LIN {X 0,Y 218.653,Z 421.951,A -85,B 0,C 180,E1 -22546.919,E2 -22546.919} C_VEL
LIN {X 0,Y 215.686,Z 434.453,A -85,B 0,C 180,E1 -22548.088,E2 -22548.088} C_VEL
LIN {X 0,Y 212.005,Z 447.131,A -85,B 0,C 180,E1 -22549.628,E2 -22549.628} C_VEL
LIN {X 0,Y 207.893,Z 459.523,A -85,B 0,C 180,E1 -22551.597,E2 -22551.597} C_VEL
LIN {X 0,Y 203.913,Z 469.49,A -85,B 0,C 180,E1 -22553.52,E2 -22553.52} C_VEL
LIN {X 0,Y 199.074,Z 480.574,A -85,B 0,C 180,E1 -22556.218,E2 -22556.218} C_VEL
LIN {X 0,Y 194.639,Z 489.759,A -85,B 0,C 180,E1 -22559.033,E2 -22559.033} C_VEL
LIN {X 0,Y 190.05,Z 498.52,A -85,B 0,C 180,E1 -22562.422,E2 -22562.422} C_VEL
LIN {X 0,Y 186.885,Z 504.847,A -85,B 0,C 180,E1 -22565.564,E2 -22565.564} C_VEL
LIN {X 0,Y 182.861,Z 511.661,A -85,B 0,C 180,E1 -22569.763,E2 -22569.763} C_VEL
LIN {X 0,Y 180.074,Z 516.84,A -85,B 0,C 180,E1 -22574.145,E2 -22574.145} C_VEL
LIN {X 0,Y 178.099,Z 520.594,A -85,B 0,C 180,E1 -22578.62,E2 -22578.62} C_VEL
LIN {X 0,Y 176.962,Z 523.045,A -85,B 0,C 180,E1 -22583.157,E2 -22583.157} C_VEL
LIN {X 0,Y 176.433,Z 524.266,A -85,B 0,C 180,E1 -22587.716,E2 -22587.716} C_VEL
LIN {X 0,Y 176.423,Z 524.285,A -85,B 0,C 180,E1 -22592.282,E2 -22592.282} C_VEL
LIN {X 0,Y 176.901,Z 523.107,A -85,B 0,C 180,E1 -22596.844,E2 -22596.844} C_VEL
LIN {X 0,Y 178.034,Z 520.699,A -85,B 0,C 180,E1 -22601.383,E2 -22601.383} C_VEL
LIN {X 0,Y 180.021,Z 516.984,A -85,B 0,C 180,E1 -22605.858,E2 -22605.858} C_VEL
LIN {X 0,Y 182.79,Z 511.867,A -85,B 0,C 180,E1 -22610.244,E2 -22610.244} C_VEL
LIN {X 0,Y 185.684,Z 506.949,A -85,B 0,C 180,E1 -22613.416,E2 -22613.416} C_VEL
LIN {X 0,Y 189.292,Z 500.114,A -85,B 0,C 180,E1 -22616.992,E2 -22616.992} C_VEL
LIN {X 0,Y 193.801,Z 491.473,A -85,B 0,C 180,E1 -22620.509,E2 -22620.509} C_VEL
LIN {X 0,Y 198.243,Z 482.622,A -85,B 0,C 180,E1 -22623.331,E2 -22623.331} C_VEL
LIN {X 0,Y 202.955,Z 471.992,A -85,B 0,C 180,E1 -22626.062,E2 -22626.062} C_VEL
LIN {X 0,Y 207.337,Z 461.314,A -85,B 0,C 180,E1 -22628.213,E2 -22628.213} C_VEL
LIN {X 0,Y 211.244,Z 450.035,A -85,B 0,C 180,E1 -22630.075,E2 -22630.075} C_VEL
LIN {X 0,Y 215.079,Z 437.178,A -85,B 0,C 180,E1 -22631.741,E2 -22631.741} C_VEL
LIN {X 0,Y 218.486,Z 423.175,A -85,B 0,C 180,E1 -22633.12,E2 -22633.12} C_VEL
LIN {X 0,Y 221.137,Z 409.142,A -85,B 0,C 180,E1 -22634.122,E2 -22634.122} C_VEL
LIN {X 0,Y 223.032,Z 394.243,A -85,B 0,C 180,E1 -22634.86,E2 -22634.86} C_VEL
LIN {X 0,Y 225.773,Z 353.828,A -85,B 0,C 180,E1 -22635.992,E2 -22635.992} C_VEL
LIN {X 0,Y 228.15,Z 314.688,A -85,B 0,C 180,E1 -22637.083,E2 -22637.083} C_VEL
LIN {X 0,Y 223.112,Z 303.279,A -85,B 0,C 180,E1 -22639.111,E2 -22639.111} C_VEL
LIN {X 0,Y 217.663,Z 292.439,A -85,B 0,C 180,E1 -22641.444,E2 -22641.444} C_VEL
LIN {X 0,Y 211.854,Z 282.14,A -85,B 0,C 180,E1 -22644.157,E2 -22644.157} C_VEL
LIN {X 0,Y 206.318,Z 273.056,A -85,B 0,C 180,E1 -22647.046,E2 -22647.046} C_VEL
LIN {X 0,Y 201.904,Z 266.645,A -85,B 0,C 180,E1 -22649.602,E2 -22649.602} C_VEL
LIN {X 0,Y 198.685,Z 262.105,A -85,B 0,C 180,E1 -22651.673,E2 -22651.673} C_VEL
LIN {X 0,Y 194.536,Z 256.634,A -85,B 0,C 180,E1 -22654.667,E2 -22654.667} C_VEL
LIN {X 0,Y 190.02,Z 250.759,A -85,B 0,C 180,E1 -22658.578,E2 -22658.578} C_VEL
LIN {X 0,Y 185.157,Z 244.692,A -85,B 0,C 180,E1 -22664.354,E2 -22664.354} C_VEL
LIN {X 0,Y 184.19,Z 241.633,A -85,B 0,C 180,E1 -22671.221,E2 -22671.221} C_VEL
LIN {X 0,Y 183.785,Z 240.861,A -85,B 0,C 180,E1 -22675.613,E2 -22675.613} C_VEL
LIN {X 0,Y 184.022,Z 240.453,A -85,B 0,C 180,E1 -22680,E2 -22680} C_VEL
LIN {X 0,Y 184.017,Z 241.278,A -85,B 0,C 180,E1 -22684.38,E2 -22684.38} C_VEL
LIN {X 0,Y 184.386,Z 242.229,A -85,B 0,C 180,E1 -22687.703,E2 -22687.703} C_VEL
LIN {X 0,Y 185.376,Z 244.972,A -85,B 0,C 180,E1 -22693.148,E2 -22693.148} C_VEL
LIN {X 0,Y 191.011,Z 251.991,A -85,B 0,C 180,E1 -22699.477,E2 -22699.477} C_VEL
LIN {X 0,Y 196.189,Z 258.564,A -85,B 0,C 180,E1 -22703.696,E2 -22703.696} C_VEL
LIN {X 0,Y 200.62,Z 264.7,A -85,B 0,C 180,E1 -22706.739,E2 -22706.739} C_VEL
LIN {X 0,Y 204.903,Z 270.949,A -85,B 0,C 180,E1 -22709.329,E2 -22709.329} C_VEL
LIN {X 0,Y 210.285,Z 279.254,A -85,B 0,C 180,E1 -22712.224,E2 -22712.224} C_VEL
LIN {X 0,Y 216.265,Z 289.677,A -85,B 0,C 180,E1 -22715.123,E2 -22715.123} C_VEL
LIN {X 0,Y 222.764,Z 302.204,A -85,B 0,C 180,E1 -22717.966,E2 -22717.966} C_VEL
LIN {X 0,Y 228.385,Z 314.765,A -85,B 0,C 180,E1 -22720.257,E2 -22720.257} C_VEL
LIN {X 0,Y 227.513,Z 328.436,A -85,B 0,C 180,E1 -22720.664,E2 -22720.664} C_VEL
LIN {X 0,Y 226.648,Z 334.283,A -85,B 0,C 180,E1 -22720.701,E2 -22720.701} C_VEL
LIN {X 0,Y 221.407,Z 353.296,A -85,B 0,C 180,E1 -22720.124,E2 -22720.124} C_VEL
LIN {X 0,Y 220.595,Z 359.139,A -85,B 0,C 180,E1 -22720.175,E2 -22720.175} C_VEL
LIN {X 0,Y 217.438,Z 402.262,A -85,B 0,C 180,E1 -22721.484,E2 -22721.484} C_VEL
LIN {X 0,Y 215.218,Z 417.373,A -85,B 0,C 180,E1 -22722.197,E2 -22722.197} C_VEL
LIN {X 0,Y 212.207,Z 432.144,A -85,B 0,C 180,E1 -22723.232,E2 -22723.232} C_VEL
LIN {X 0,Y 208.441,Z 446.371,A -85,B 0,C 180,E1 -22724.582,E2 -22724.582} C_VEL
LIN {X 0,Y 204.284,Z 459.462,A -85,B 0,C 180,E1 -22726.219,E2 -22726.219} C_VEL
LIN {X 0,Y 199.49,Z 472.49,A -85,B 0,C 180,E1 -22728.322,E2 -22728.322} C_VEL
LIN {X 0,Y 194.43,Z 484.437,A -85,B 0,C 180,E1 -22730.762,E2 -22730.762} C_VEL
LIN {X 0,Y 189.385,Z 495.303,A -85,B 0,C 180,E1 -22733.578,E2 -22733.578} C_VEL
LIN {X 0,Y 184.246,Z 505.783,A -85,B 0,C 180,E1 -22737.053,E2 -22737.053} C_VEL
LIN {X 0,Y 179.923,Z 514.522,A -85,B 0,C 180,E1 -22740.775,E2 -22740.775} C_VEL
LIN {X 0,Y 176.589,Z 520.747,A -85,B 0,C 180,E1 -22744.039,E2 -22744.039} C_VEL
LIN {X 0,Y 173.204,Z 527.526,A -85,B 0,C 180,E1 -22748.582,E2 -22748.582} C_VEL
LIN {X 0,Y 170.848,Z 532.779,A -85,B 0,C 180,E1 -22753.266,E2 -22753.266} C_VEL
LIN {X 0,Y 169.447,Z 536.638,A -85,B 0,C 180,E1 -22758.032,E2 -22758.032} C_VEL
LIN {X 0,Y 169.001,Z 539.191,A -85,B 0,C 180,E1 -22762.834,E2 -22762.834} C_VEL
LIN {X 0,Y 169.058,Z 540.184,A -85,B 0,C 180,E1 -22766.121,E2 -22766.121} C_VEL
LIN {X 0,Y 169.244,Z 540.643,A -85,B 0,C 180,E1 -22770.001,E2 -22770.001} C_VEL
LIN {X 0,Y 169.019,Z 539.974,A -85,B 0,C 180,E1 -22774.771,E2 -22774.771} C_VEL
LIN {X 0,Y 169.119,Z 538.035,A -85,B 0,C 180,E1 -22779.569,E2 -22779.569} C_VEL
LIN {X 0,Y 170.023,Z 534.819,A -85,B 0,C 180,E1 -22784.361,E2 -22784.361} C_VEL
LIN {X 0,Y 171.937,Z 530.261,A -85,B 0,C 180,E1 -22789.088,E2 -22789.088} C_VEL
LIN {X 0,Y 174.79,Z 524.236,A -85,B 0,C 180,E1 -22793.709,E2 -22793.709} C_VEL
LIN {X 0,Y 178.702,Z 516.59,A -85,B 0,C 180,E1 -22798.161,E2 -22798.161} C_VEL
LIN {X 0,Y 182.96,Z 508.339,A -85,B 0,C 180,E1 -22801.883,E2 -22801.883} C_VEL
LIN {X 0,Y 187.036,Z 499.871,A -85,B 0,C 180,E1 -22804.962,E2 -22804.962} C_VEL
LIN {X 0,Y 191.832,Z 489.882,A -85,B 0,C 180,E1 -22807.855,E2 -22807.855} C_VEL
LIN {X 0,Y 196.172,Z 480.085,A -85,B 0,C 180,E1 -22810.156,E2 -22810.156} C_VEL
LIN {X 0,Y 201.233,Z 467.679,A -85,B 0,C 180,E1 -22812.461,E2 -22812.461} C_VEL
LIN {X 0,Y 205.793,Z 454.351,A -85,B 0,C 180,E1 -22814.433,E2 -22814.433} C_VEL
LIN {X 0,Y 209.977,Z 440.166,A -85,B 0,C 180,E1 -22816.023,E2 -22816.023} C_VEL
LIN {X 0,Y 213.256,Z 426.593,A -85,B 0,C 180,E1 -22817.161,E2 -22817.161} C_VEL
LIN {X 0,Y 215.943,Z 412.233,A -85,B 0,C 180,E1 -22818.028,E2 -22818.028} C_VEL
LIN {X 0,Y 217.721,Z 397.26,A -85,B 0,C 180,E1 -22818.661,E2 -22818.661} C_VEL
LIN {X 0,Y 223.372,Z 317.086,A -85,B 0,C 180,E1 -22821.004,E2 -22821.004} C_VEL
LIN {X 0,Y 218.369,Z 305.775,A -85,B 0,C 180,E1 -22823.171,E2 -22823.171} C_VEL
LIN {X 0,Y 212.544,Z 294.337,A -85,B 0,C 180,E1 -22825.869,E2 -22825.869} C_VEL
LIN {X 0,Y 206.67,Z 283.81,A -85,B 0,C 180,E1 -22828.884,E2 -22828.884} C_VEL
LIN {X 0,Y 200.82,Z 274.478,A -85,B 0,C 180,E1 -22832.273,E2 -22832.273} C_VEL
LIN {X 0,Y 196.8,Z 268.677,A -85,B 0,C 180,E1 -22834.908,E2 -22834.908} C_VEL
LIN {X 0,Y 192.99,Z 263.374,A -85,B 0,C 180,E1 -22837.748,E2 -22837.748} C_VEL
LIN {X 0,Y 188.292,Z 257.278,A -85,B 0,C 180,E1 -22841.925,E2 -22841.925} C_VEL
LIN {X 0,Y 183.747,Z 251.493,A -85,B 0,C 180,E1 -22847.296,E2 -22847.296} C_VEL
LIN {X 0,Y 180.186,Z 247.396,A -85,B 0,C 180,E1 -22853.991,E2 -22853.991} C_VEL
LIN {X 0,Y 178.998,Z 245.415,A -85,B 0,C 180,E1 -22860,E2 -22860} C_VEL
LIN {X 0,Y 179.647,Z 246.794,A -85,B 0,C 180,E1 -22867.305,E2 -22867.305} C_VEL
LIN {X 0,Y 180.952,Z 248.541,A -85,B 0,C 180,E1 -22870.915,E2 -22870.915} C_VEL
LIN {X 0,Y 184.159,Z 252.061,A -85,B 0,C 180,E1 -22876.256,E2 -22876.256} C_VEL
LIN {X 0,Y 189.107,Z 258.285,A -85,B 0,C 180,E1 -22881.817,E2 -22881.817} C_VEL
LIN {X 0,Y 193.938,Z 264.803,A -85,B 0,C 180,E1 -22885.941,E2 -22885.941} C_VEL
LIN {X 0,Y 197.828,Z 270.248,A -85,B 0,C 180,E1 -22888.732,E2 -22888.732} C_VEL
LIN {X 0,Y 201.626,Z 275.937,A -85,B 0,C 180,E1 -22891.152,E2 -22891.152} C_VEL
LIN {X 0,Y 204.826,Z 281.081,A -85,B 0,C 180,E1 -22893.019,E2 -22893.019} C_VEL
LIN {X 0,Y 209.64,Z 289.143,A -85,B 0,C 180,E1 -22895.577,E2 -22895.577} C_VEL
LIN {X 0,Y 215.341,Z 299.835,A -85,B 0,C 180,E1 -22898.324,E2 -22898.324} C_VEL
LIN {X 0,Y 220.901,Z 311.625,A -85,B 0,C 180,E1 -22900.784,E2 -22900.784} C_VEL
LIN {X 0,Y 223.174,Z 317.039,A -85,B 0,C 180,E1 -22901.746,E2 -22901.746} C_VEL
LIN {X 0,Y 218.401,Z 390.017,A -85,B 0,C 180,E1 -22903.783,E2 -22903.783} C_VEL
LIN {X 0,Y 216.873,Z 403.965,A -85,B 0,C 180,E1 -22904.381,E2 -22904.381} C_VEL
LIN {X 0,Y 214.562,Z 417.52,A -85,B 0,C 180,E1 -22905.232,E2 -22905.232} C_VEL
LIN {X 0,Y 211.514,Z 431.044,A -85,B 0,C 180,E1 -22906.412,E2 -22906.412} C_VEL
LIN {X 0,Y 207.952,Z 443.347,A -85,B 0,C 180,E1 -22907.79,E2 -22907.79} C_VEL
LIN {X 0,Y 203.803,Z 456.167,A -85,B 0,C 180,E1 -22909.715,E2 -22909.715} C_VEL
LIN {X 0,Y 199.184,Z 467.757,A -85,B 0,C 180,E1 -22911.868,E2 -22911.868} C_VEL
LIN {X 0,Y 194.87,Z 477.443,A -85,B 0,C 180,E1 -22914.122,E2 -22914.122} C_VEL
LIN {X 0,Y 190.135,Z 487.191,A -85,B 0,C 180,E1 -22916.961,E2 -22916.961} C_VEL
LIN {X 0,Y 185.039,Z 496.568,A -85,B 0,C 180,E1 -22920.412,E2 -22920.412} C_VEL
LIN {X 0,Y 182.045,Z 502.219,A -85,B 0,C 180,E1 -22923.023,E2 -22923.023} C_VEL
LIN {X 0,Y 178.223,Z 508.808,A -85,B 0,C 180,E1 -22926.775,E2 -22926.775} C_VEL
LIN {X 0,Y 175.398,Z 513.398,A -85,B 0,C 180,E1 -22930.087,E2 -22930.087} C_VEL
LIN {X 0,Y 172.65,Z 518.208,A -85,B 0,C 180,E1 -22934.657,E2 -22934.657} C_VEL
LIN {X 0,Y 171.147,Z 520.928,A -85,B 0,C 180,E1 -22938.151,E2 -22938.151} C_VEL
LIN {X 0,Y 169.926,Z 523.378,A -85,B 0,C 180,E1 -22942.872,E2 -22942.872} C_VEL
LIN {X 0,Y 169.361,Z 524.599,A -85,B 0,C 180,E1 -22947.621,E2 -22947.621} C_VEL
LIN {X 0,Y 169.35,Z 524.617,A -85,B 0,C 180,E1 -22952.378,E2 -22952.378} C_VEL
LIN {X 0,Y 169.867,Z 523.44,A -85,B 0,C 180,E1 -22957.129,E2 -22957.129} C_VEL
LIN {X 0,Y 171.094,Z 521.031,A -85,B 0,C 180,E1 -22961.851,E2 -22961.851} C_VEL
LIN {X 0,Y 173.21,Z 517.317,A -85,B 0,C 180,E1 -22966.499,E2 -22966.499} C_VEL
LIN {X 0,Y 176.139,Z 512.202,A -85,B 0,C 180,E1 -22971.044,E2 -22971.044} C_VEL
LIN {X 0,Y 180.307,Z 505.471,A -85,B 0,C 180,E1 -22975.387,E2 -22975.387} C_VEL
LIN {X 0,Y 183.657,Z 499.253,A -85,B 0,C 180,E1 -22978.574,E2 -22978.574} C_VEL
LIN {X 0,Y 188.482,Z 490.486,A -85,B 0,C 180,E1 -22982.095,E2 -22982.095} C_VEL
LIN {X 0,Y 193.142,Z 481.374,A -85,B 0,C 180,E1 -22984.966,E2 -22984.966} C_VEL
LIN {X 0,Y 198.229,Z 470.422,A -85,B 0,C 180,E1 -22987.702,E2 -22987.702} C_VEL
LIN {X 0,Y 202.78,Z 459.374,A -85,B 0,C 180,E1 -22989.878,E2 -22989.878} C_VEL
LIN {X 0,Y 206.84,Z 447.571,A -85,B 0,C 180,E1 -22991.77,E2 -22991.77} C_VEL
LIN {X 0,Y 210.372,Z 435.877,A -85,B 0,C 180,E1 -22993.222,E2 -22993.222} C_VEL
LIN {X 0,Y 213.659,Z 422.571,A -85,B 0,C 180,E1 -22994.509,E2 -22994.509} C_VEL
LIN {X 0,Y 216.392,Z 408.255,A -85,B 0,C 180,E1 -22995.519,E2 -22995.519} C_VEL
LIN {X 0,Y 218.289,Z 393.244,A -85,B 0,C 180,E1 -22996.246,E2 -22996.246} C_VEL
LIN {X 0,Y 223.382,Z 317.653,A -85,B 0,C 180,E1 -22998.341,E2 -22998.341} C_VEL
LIN {X 0,Y 221.754,Z 313.323,A -85,B 0,C 180,E1 -22999.049,E2 -22999.049} C_VEL
LIN {X 0,Y 216.111,Z 301.185,A -85,B 0,C 180,E1 -23001.528,E2 -23001.528} C_VEL
LIN {X 0,Y 210.735,Z 291.036,A -85,B 0,C 180,E1 -23004.087,E2 -23004.087} C_VEL
LIN {X 0,Y 205.419,Z 281.911,A -85,B 0,C 180,E1 -23006.883,E2 -23006.883} C_VEL
LIN {X 0,Y 202.152,Z 276.744,A -85,B 0,C 180,E1 -23008.77,E2 -23008.77} C_VEL
LIN {X 0,Y 199.374,Z 272.502,A -85,B 0,C 180,E1 -23010.506,E2 -23010.506} C_VEL
LIN {X 0,Y 196.518,Z 268.359,A -85,B 0,C 180,E1 -23012.439,E2 -23012.439} C_VEL
LIN {X 0,Y 192.683,Z 263.101,A -85,B 0,C 180,E1 -23015.343,E2 -23015.343} C_VEL
LIN {X 0,Y 188.388,Z 257.316,A -85,B 0,C 180,E1 -23019.242,E2 -23019.242} C_VEL
LIN {X 0,Y 183.605,Z 251.366,A -85,B 0,C 180,E1 -23025.026,E2 -23025.026} C_VEL
LIN {X 0,Y 180.122,Z 247.334,A -85,B 0,C 180,E1 -23032.151,E2 -23032.151} C_VEL
LIN {X 0,Y 179.203,Z 245.923,A -85,B 0,C 180,E1 -23037.752,E2 -23037.752} C_VEL
LIN {X 0,Y 179.304,Z 245.874,A -85,B 0,C 180,E1 -23040.561,E2 -23040.561} C_VEL
LIN {X 0,Y 180.737,Z 247.995,A -85,B 0,C 180,E1 -23046.699,E2 -23046.699} C_VEL
LIN {X 0,Y 184.196,Z 252.048,A -85,B 0,C 180,E1 -23052.953,E2 -23052.953} C_VEL
LIN {X 0,Y 189.45,Z 258.718,A -85,B 0,C 180,E1 -23058.941,E2 -23058.941} C_VEL
LIN {X 0,Y 194.155,Z 264.882,A -85,B 0,C 180,E1 -23062.95,E2 -23062.95} C_VEL
LIN {X 0,Y 198.301,Z 270.822,A -85,B 0,C 180,E1 -23065.943,E2 -23065.943} C_VEL
LIN {X 0,Y 202.203,Z 276.675,A -85,B 0,C 180,E1 -23068.426,E2 -23068.426} C_VEL
LIN {X 0,Y 207.154,Z 284.521,A -85,B 0,C 180,E1 -23071.239,E2 -23071.239} C_VEL
LIN {X 0,Y 212.297,Z 293.725,A -85,B 0,C 180,E1 -23073.89,E2 -23073.89} C_VEL
LIN {X 0,Y 218.305,Z 305.56,A -85,B 0,C 180,E1 -23076.697,E2 -23076.697} C_VEL
LIN {X 0,Y 223.073,Z 316.161,A -85,B 0,C 180,E1 -23078.768,E2 -23078.768} C_VEL
LIN {X 0,Y 223.587,Z 317.439,A -85,B 0,C 180,E1 -23078.987,E2 -23078.987} C_VEL
LIN {X 0,Y 220.595,Z 359.139,A -85,B 0,C 180,E1 -23080.175,E2 -23080.175} C_VEL
LIN {X 0,Y 219.799,Z 364.986,A -85,B 0,C 180,E1 -23080.23,E2 -23080.23} C_VEL
LIN {X 0,Y 214.663,Z 384.044,A -85,B 0,C 180,E1 -23079.646,E2 -23079.646} C_VEL
LIN {X 0,Y 213.772,Z 389.899,A -85,B 0,C 180,E1 -23079.673,E2 -23079.673} C_VEL
LIN {X 0,Y 212.203,Z 405.842,A -85,B 0,C 180,E1 -23080.223,E2 -23080.223} C_VEL
LIN {X 0,Y 209.819,Z 420.533,A -85,B 0,C 180,E1 -23081.003,E2 -23081.003} C_VEL
LIN {X 0,Y 206.554,Z 435.008,A -85,B 0,C 180,E1 -23082.085,E2 -23082.085} C_VEL
LIN {X 0,Y 202.402,Z 449.455,A -85,B 0,C 180,E1 -23083.546,E2 -23083.546} C_VEL
LIN {X 0,Y 197.967,Z 462.499,A -85,B 0,C 180,E1 -23085.308,E2 -23085.308} C_VEL
LIN {X 0,Y 192.724,Z 475.641,A -85,B 0,C 180,E1 -23087.576,E2 -23087.576} C_VEL
LIN {X 0,Y 188.041,Z 486.039,A -85,B 0,C 180,E1 -23089.857,E2 -23089.857} C_VEL
LIN {X 0,Y 182.835,Z 496.593,A -85,B 0,C 180,E1 -23092.743,E2 -23092.743} C_VEL
LIN {X 0,Y 177.535,Z 506.854,A -85,B 0,C 180,E1 -23096.345,E2 -23096.345} C_VEL
LIN {X 0,Y 173.076,Z 515.316,A -85,B 0,C 180,E1 -23100.171,E2 -23100.171} C_VEL
LIN {X 0,Y 169.137,Z 522.26,A -85,B 0,C 180,E1 -23104.134,E2 -23104.134} C_VEL
LIN {X 0,Y 165.781,Z 528.62,A -85,B 0,C 180,E1 -23108.851,E2 -23108.851} C_VEL
LIN {X 0,Y 163.504,Z 533.547,A -85,B 0,C 180,E1 -23113.777,E2 -23113.777} C_VEL
LIN {X 0,Y 162.446,Z 536.302,A -85,B 0,C 180,E1 -23117.508,E2 -23117.508} C_VEL
LIN {X 0,Y 161.916,Z 538.856,A -85,B 0,C 180,E1 -23122.519,E2 -23122.519} C_VEL
LIN {X 0,Y 161.964,Z 539.94,A -85,B 0,C 180,E1 -23126.394,E2 -23126.394} C_VEL
LIN {X 0,Y 162.163,Z 540.31,A -85,B 0,C 180,E1 -23130.001,E2 -23130.001} C_VEL
LIN {X 0,Y 161.926,Z 539.64,A -85,B 0,C 180,E1 -23134.981,E2 -23134.981} C_VEL
LIN {X 0,Y 162.073,Z 537.699,A -85,B 0,C 180,E1 -23139.989,E2 -23139.989} C_VEL
LIN {X 0,Y 163.105,Z 534.482,A -85,B 0,C 180,E1 -23144.984,E2 -23144.984} C_VEL
LIN {X 0,Y 165.149,Z 529.92,A -85,B 0,C 180,E1 -23149.905,E2 -23149.905} C_VEL
LIN {X 0,Y 168.224,Z 523.893,A -85,B 0,C 180,E1 -23154.695,E2 -23154.695} C_VEL
LIN {X 0,Y 172.43,Z 516.245,A -85,B 0,C 180,E1 -23159.282,E2 -23159.282} C_VEL
LIN {X 0,Y 176.905,Z 507.987,A -85,B 0,C 180,E1 -23163.111,E2 -23163.111} C_VEL
LIN {X 0,Y 181.211,Z 499.511,A -85,B 0,C 180,E1 -23166.26,E2 -23166.26} C_VEL
LIN {X 0,Y 186.245,Z 489.511,A -85,B 0,C 180,E1 -23169.203,E2 -23169.203} C_VEL
LIN {X 0,Y 190.781,Z 479.697,A -85,B 0,C 180,E1 -23171.536,E2 -23171.536} C_VEL
LIN {X 0,Y 195.863,Z 467.673,A -85,B 0,C 180,E1 -23173.804,E2 -23173.804} C_VEL
LIN {X 0,Y 200.244,Z 455.488,A -85,B 0,C 180,E1 -23175.652,E2 -23175.652} C_VEL
LIN {X 0,Y 204.557,Z 441.655,A -85,B 0,C 180,E1 -23177.255,E2 -23177.255} C_VEL
LIN {X 0,Y 208.195,Z 427.299,A -85,B 0,C 180,E1 -23178.502,E2 -23178.502} C_VEL
LIN {X 0,Y 211.107,Z 412.389,A -85,B 0,C 180,E1 -23179.416,E2 -23179.416} C_VEL
LIN {X 0,Y 212.994,Z 397.081,A -85,B 0,C 180,E1 -23180.069,E2 -23180.069} C_VEL
LIN {X 0,Y 218.623,Z 320.887,A -85,B 0,C 180,E1 -23182.289,E2 -23182.289} C_VEL
LIN {X 0,Y 218.512,Z 319.369,A -85,B 0,C 180,E1 -23182.404,E2 -23182.404} C_VEL
LIN {X 0,Y 213.696,Z 308.33,A -85,B 0,C 180,E1 -23184.647,E2 -23184.647} C_VEL
LIN {X 0,Y 207.815,Z 296.712,A -85,B 0,C 180,E1 -23187.587,E2 -23187.587} C_VEL
LIN {X 0,Y 202.687,Z 287.637,A -85,B 0,C 180,E1 -23190.43,E2 -23190.43} C_VEL
LIN {X 0,Y 197.872,Z 279.793,A -85,B 0,C 180,E1 -23193.43,E2 -23193.43} C_VEL
LIN {X 0,Y 194.389,Z 274.611,A -85,B 0,C 180,E1 -23195.859,E2 -23195.859} C_VEL
LIN {X 0,Y 190.689,Z 269.247,A -85,B 0,C 180,E1 -23198.799,E2 -23198.799} C_VEL
LIN {X 0,Y 186.777,Z 263.975,A -85,B 0,C 180,E1 -23202.481,E2 -23202.481} C_VEL
LIN {X 0,Y 182.314,Z 258.136,A -85,B 0,C 180,E1 -23208.042,E2 -23208.042} C_VEL
LIN {X 0,Y 179.118,Z 254.274,A -85,B 0,C 180,E1 -23214.519,E2 -23214.519} C_VEL
LIN {X 0,Y 178.081,Z 252.48,A -85,B 0,C 180,E1 -23220,E2 -23220} C_VEL
LIN {X 0,Y 178.774,Z 253.873,A -85,B 0,C 180,E1 -23227.305,E2 -23227.305} C_VEL
LIN {X 0,Y 180.084,Z 255.735,A -85,B 0,C 180,E1 -23230.968,E2 -23230.968} C_VEL
LIN {X 0,Y 182.873,Z 258.894,A -85,B 0,C 180,E1 -23235.749,E2 -23235.749} C_VEL
LIN {X 0,Y 187.526,Z 264.951,A -85,B 0,C 180,E1 -23241.22,E2 -23241.22} C_VEL
LIN {X 0,Y 191.964,Z 271.147,A -85,B 0,C 180,E1 -23245.189,E2 -23245.189} C_VEL
LIN {X 0,Y 195.6,Z 276.411,A -85,B 0,C 180,E1 -23247.932,E2 -23247.932} C_VEL
LIN {X 0,Y 199.182,Z 282.012,A -85,B 0,C 180,E1 -23250.336,E2 -23250.336} C_VEL
LIN {X 0,Y 203.81,Z 289.593,A -85,B 0,C 180,E1 -23253.107,E2 -23253.107} C_VEL
LIN {X 0,Y 209.266,Z 299.594,A -85,B 0,C 180,E1 -23256.032,E2 -23256.032} C_VEL
LIN {X 0,Y 214.291,Z 309.868,A -85,B 0,C 180,E1 -23258.483,E2 -23258.483} C_VEL
LIN {X 0,Y 218.504,Z 319.642,A -85,B 0,C 180,E1 -23260.411,E2 -23260.411} C_VEL
LIN {X 0,Y 213.307,Z 394.059,A -85,B 0,C 180,E1 -23262.513,E2 -23262.513} C_VEL
LIN {X 0,Y 211.322,Z 408.826,A -85,B 0,C 180,E1 -23263.235,E2 -23263.235} C_VEL
LIN {X 0,Y 208.843,Z 421.903,A -85,B 0,C 180,E1 -23264.175,E2 -23264.175} C_VEL
LIN {X 0,Y 205.391,Z 435.394,A -85,B 0,C 180,E1 -23265.455,E2 -23265.455} C_VEL
LIN {X 0,Y 201.737,Z 447.067,A -85,B 0,C 180,E1 -23266.885,E2 -23266.885} C_VEL
LIN {X 0,Y 197.509,Z 459.131,A -85,B 0,C 180,E1 -23268.83,E2 -23268.83} C_VEL
LIN {X 0,Y 192.701,Z 470.26,A -85,B 0,C 180,E1 -23271.014,E2 -23271.014} C_VEL
LIN {X 0,Y 187.451,Z 481.298,A -85,B 0,C 180,E1 -23273.807,E2 -23273.807} C_VEL
LIN {X 0,Y 182.632,Z 490.466,A -85,B 0,C 180,E1 -23276.745,E2 -23276.745} C_VEL
LIN {X 0,Y 177.404,Z 499.509,A -85,B 0,C 180,E1 -23280.447,E2 -23280.447} C_VEL
LIN {X 0,Y 174.064,Z 505.531,A -85,B 0,C 180,E1 -23283.631,E2 -23283.631} C_VEL
LIN {X 0,Y 169.593,Z 512.338,A -85,B 0,C 180,E1 -23288.101,E2 -23288.101} C_VEL
LIN {X 0,Y 166.454,Z 517.51,A -85,B 0,C 180,E1 -23292.809,E2 -23292.809} C_VEL
LIN {X 0,Y 164.197,Z 521.262,A -85,B 0,C 180,E1 -23297.642,E2 -23297.642} C_VEL
LIN {X 0,Y 162.896,Z 523.711,A -85,B 0,C 180,E1 -23302.562,E2 -23302.562} C_VEL
LIN {X 0,Y 162.291,Z 524.931,A -85,B 0,C 180,E1 -23307.517,E2 -23307.517} C_VEL
LIN {X 0,Y 162.279,Z 524.949,A -85,B 0,C 180,E1 -23312.481,E2 -23312.481} C_VEL
LIN {X 0,Y 162.822,Z 523.772,A -85,B 0,C 180,E1 -23317.439,E2 -23317.439} C_VEL
LIN {X 0,Y 164.153,Z 521.363,A -85,B 0,C 180,E1 -23322.36,E2 -23322.36} C_VEL
LIN {X 0,Y 166.409,Z 517.65,A -85,B 0,C 180,E1 -23327.194,E2 -23327.194} C_VEL
LIN {X 0,Y 169.532,Z 512.537,A -85,B 0,C 180,E1 -23331.906,E2 -23331.906} C_VEL
LIN {X 0,Y 173.904,Z 505.811,A -85,B 0,C 180,E1 -23336.393,E2 -23336.393} C_VEL
LIN {X 0,Y 177.459,Z 499.594,A -85,B 0,C 180,E1 -23339.67,E2 -23339.67} C_VEL
LIN {X 0,Y 181.731,Z 492.167,A -85,B 0,C 180,E1 -23342.779,E2 -23342.779} C_VEL
LIN {X 0,Y 186.557,Z 483.334,A -85,B 0,C 180,E1 -23345.725,E2 -23345.725} C_VEL
LIN {X 0,Y 191.699,Z 472.729,A -85,B 0,C 180,E1 -23348.552,E2 -23348.552} C_VEL
LIN {X 0,Y 196.423,Z 462.089,A -85,B 0,C 180,E1 -23350.765,E2 -23350.765} C_VEL
LIN {X 0,Y 201.199,Z 449.19,A -85,B 0,C 180,E1 -23352.93,E2 -23352.93} C_VEL
LIN {X 0,Y 204.757,Z 438.094,A -85,B 0,C 180,E1 -23354.372,E2 -23354.372} C_VEL
LIN {X 0,Y 208.4,Z 424.227,A -85,B 0,C 180,E1 -23355.775,E2 -23355.775} C_VEL
LIN {X 0,Y 211.365,Z 409.663,A -85,B 0,C 180,E1 -23356.837,E2 -23356.837} C_VEL
LIN {X 0,Y 213.301,Z 395.573,A -85,B 0,C 180,E1 -23357.557,E2 -23357.557} C_VEL
LIN {X 0,Y 215.274,Z 370.403,A -85,B 0,C 180,E1 -23358.301,E2 -23358.301} C_VEL
LIN {X 0,Y 218.632,Z 319.621,A -85,B 0,C 180,E1 -23359.733,E2 -23359.733} C_VEL
LIN {X 0,Y 213.859,Z 308.783,A -85,B 0,C 180,E1 -23361.924,E2 -23361.924} C_VEL
LIN {X 0,Y 209.018,Z 299.045,A -85,B 0,C 180,E1 -23364.306,E2 -23364.306} C_VEL
LIN {X 0,Y 203.547,Z 289.054,A -85,B 0,C 180,E1 -23367.277,E2 -23367.277} C_VEL
LIN {X 0,Y 199.883,Z 283.063,A -85,B 0,C 180,E1 -23369.471,E2 -23369.471} C_VEL
LIN {X 0,Y 197.083,Z 278.625,A -85,B 0,C 180,E1 -23371.306,E2 -23371.306} C_VEL
LIN {X 0,Y 194.001,Z 274.072,A -85,B 0,C 180,E1 -23373.51,E2 -23373.51} C_VEL
LIN {X 0,Y 190.781,Z 269.485,A -85,B 0,C 180,E1 -23376.095,E2 -23376.095} C_VEL
LIN {X 0,Y 186.775,Z 263.929,A -85,B 0,C 180,E1 -23379.918,E2 -23379.918} C_VEL
LIN {X 0,Y 182.396,Z 258.198,A -85,B 0,C 180,E1 -23385.495,E2 -23385.495} C_VEL
LIN {X 0,Y 179.095,Z 254.229,A -85,B 0,C 180,E1 -23392.672,E2 -23392.672} C_VEL
LIN {X 0,Y 178.319,Z 252.88,A -85,B 0,C 180,E1 -23398.87,E2 -23398.87} C_VEL
LIN {X 0,Y 178.475,Z 253.051,A -85,B 0,C 180,E1 -23401.128,E2 -23401.128} C_VEL
LIN {X 0,Y 180.097,Z 255.484,A -85,B 0,C 180,E1 -23407.315,E2 -23407.315} C_VEL
LIN {X 0,Y 182.943,Z 258.872,A -85,B 0,C 180,E1 -23412.479,E2 -23412.479} C_VEL
LIN {X 0,Y 187.78,Z 265.252,A -85,B 0,C 180,E1 -23418.267,E2 -23418.267} C_VEL
LIN {X 0,Y 192.158,Z 271.248,A -85,B 0,C 180,E1 -23422.197,E2 -23422.197} C_VEL
LIN {X 0,Y 196.105,Z 277.061,A -85,B 0,C 180,E1 -23425.187,E2 -23425.187} C_VEL
LIN {X 0,Y 199.781,Z 282.785,A -85,B 0,C 180,E1 -23427.645,E2 -23427.645} C_VEL
LIN {X 0,Y 204.393,Z 290.409,A -85,B 0,C 180,E1 -23430.404,E2 -23430.404} C_VEL
LIN {X 0,Y 209.471,Z 299.792,A -85,B 0,C 180,E1 -23433.15,E2 -23433.15} C_VEL
LIN {X 0,Y 215.484,Z 312.039,A -85,B 0,C 180,E1 -23436.087,E2 -23436.087} C_VEL
LIN {X 0,Y 218.864,Z 319.934,A -85,B 0,C 180,E1 -23437.641,E2 -23437.641} C_VEL
LIN {X 0,Y 213.772,Z 389.899,A -85,B 0,C 180,E1 -23439.673,E2 -23439.673} C_VEL
LIN {X 0,Y 212.855,Z 395.727,A -85,B 0,C 180,E1 -23439.707,E2 -23439.707} C_VEL
LIN {X 0,Y 210,Z 405.17,A -85,B 0,C 180,E1 -23439.486,E2 -23439.486} C_VEL
LIN {X 0,Y 207.35,Z 412.638,A -85,B 0,C 180,E1 -23439.347,E2 -23439.347} C_VEL
LIN {X 0,Y 205.623,Z 418.295,A -85,B 0,C 180,E1 -23439.432,E2 -23439.432} C_VEL
LIN {X 0,Y 205.177,Z 420.192,A -85,B 0,C 180,E1 -23439.527,E2 -23439.527} C_VEL
LIN {X 0,Y 201.845,Z 434.48,A -85,B 0,C 180,E1 -23440.583,E2 -23440.583} C_VEL
LIN {X 0,Y 198.127,Z 447.22,A -85,B 0,C 180,E1 -23441.85,E2 -23441.85} C_VEL
LIN {X 0,Y 193.728,Z 459.909,A -85,B 0,C 180,E1 -23443.487,E2 -23443.487} C_VEL
LIN {X 0,Y 188.553,Z 472.889,A -85,B 0,C 180,E1 -23445.665,E2 -23445.665} C_VEL
LIN {X 0,Y 183.527,Z 483.686,A -85,B 0,C 180,E1 -23447.923,E2 -23447.923} C_VEL
LIN {X 0,Y 178.047,Z 494.58,A -85,B 0,C 180,E1 -23450.836,E2 -23450.836} C_VEL
LIN {X 0,Y 172.956,Z 504.021,A -85,B 0,C 180,E1 -23454.045,E2 -23454.045} C_VEL
LIN {X 0,Y 168.169,Z 512.688,A -85,B 0,C 180,E1 -23457.804,E2 -23457.804} C_VEL
LIN {X 0,Y 163.767,Z 520.063,A -85,B 0,C 180,E1 -23461.833,E2 -23461.833} C_VEL
LIN {X 0,Y 159.903,Z 526.848,A -85,B 0,C 180,E1 -23466.7,E2 -23466.7} C_VEL
LIN {X 0,Y 157.131,Z 532.103,A -85,B 0,C 180,E1 -23471.756,E2 -23471.756} C_VEL
LIN {X 0,Y 155.444,Z 535.966,A -85,B 0,C 180,E1 -23476.936,E2 -23476.936} C_VEL
LIN {X 0,Y 154.834,Z 538.521,A -85,B 0,C 180,E1 -23482.175,E2 -23482.175} C_VEL
LIN {X 0,Y 154.895,Z 539.671,A -85,B 0,C 180,E1 -23486.551,E2 -23486.551} C_VEL
LIN {X 0,Y 155.063,Z 539.977,A -85,B 0,C 180,E1 -23490.001,E2 -23490.001} C_VEL
LIN {X 0,Y 154.836,Z 539.306,A -85,B 0,C 180,E1 -23495.209,E2 -23495.209} C_VEL
LIN {X 0,Y 155.019,Z 537.362,A -85,B 0,C 180,E1 -23500.449,E2 -23500.449} C_VEL
LIN {X 0,Y 156.203,Z 534.145,A -85,B 0,C 180,E1 -23505.662,E2 -23505.662} C_VEL
LIN {X 0,Y 158.382,Z 529.579,A -85,B 0,C 180,E1 -23510.794,E2 -23510.794} C_VEL
LIN {X 0,Y 161.701,Z 523.549,A -85,B 0,C 180,E1 -23515.762,E2 -23515.762} C_VEL
LIN {X 0,Y 165.56,Z 516.928,A -85,B 0,C 180,E1 -23519.92,E2 -23519.92} C_VEL
LIN {X 0,Y 170.153,Z 508.988,A -85,B 0,C 180,E1 -23523.835,E2 -23523.835} C_VEL
LIN {X 0,Y 174.653,Z 500.66,A -85,B 0,C 180,E1 -23527.128,E2 -23527.128} C_VEL
LIN {X 0,Y 179.821,Z 490.943,A -85,B 0,C 180,E1 -23530.157,E2 -23530.157} C_VEL
LIN {X 0,Y 184.979,Z 480.387,A -85,B 0,C 180,E1 -23532.776,E2 -23532.776} C_VEL
LIN {X 0,Y 190.267,Z 468.542,A -85,B 0,C 180,E1 -23535.073,E2 -23535.073} C_VEL
LIN {X 0,Y 194.792,Z 456.626,A -85,B 0,C 180,E1 -23536.938,E2 -23536.938} C_VEL
LIN {X 0,Y 199.223,Z 443.141,A -85,B 0,C 180,E1 -23538.559,E2 -23538.559} C_VEL
LIN {X 0,Y 202.936,Z 429.297,A -85,B 0,C 180,E1 -23539.824,E2 -23539.824} C_VEL
LIN {X 0,Y 205.91,Z 415.246,A -85,B 0,C 180,E1 -23540.747,E2 -23540.747} C_VEL
LIN {X 0,Y 207.976,Z 401.335,A -85,B 0,C 180,E1 -23541.383,E2 -23541.383} C_VEL
LIN {X 0,Y 214.083,Z 322.387,A -85,B 0,C 180,E1 -23543.726,E2 -23543.726} C_VEL
LIN {X 0,Y 209.417,Z 311.667,A -85,B 0,C 180,E1 -23546.044,E2 -23546.044} C_VEL
LIN {X 0,Y 204.196,Z 301.094,A -85,B 0,C 180,E1 -23548.846,E2 -23548.846} C_VEL
LIN {X 0,Y 199.281,Z 292.15,A -85,B 0,C 180,E1 -23551.771,E2 -23551.771} C_VEL
LIN {X 0,Y 194.881,Z 284.859,A -85,B 0,C 180,E1 -23554.715,E2 -23554.715} C_VEL
LIN {X 0,Y 191.992,Z 280.462,A -85,B 0,C 180,E1 -23556.867,E2 -23556.867} C_VEL
LIN {X 0,Y 188.785,Z 275.626,A -85,B 0,C 180,E1 -23559.574,E2 -23559.574} C_VEL
LIN {X 0,Y 185.197,Z 270.584,A -85,B 0,C 180,E1 -23563.134,E2 -23563.134} C_VEL
LIN {X 0,Y 181.262,Z 265.148,A -85,B 0,C 180,E1 -23568.255,E2 -23568.255} C_VEL
LIN {X 0,Y 178.091,Z 261.152,A -85,B 0,C 180,E1 -23574.981,E2 -23574.981} C_VEL
LIN {X 0,Y 177.212,Z 259.551,A -85,B 0,C 180,E1 -23580,E2 -23580} C_VEL
LIN {X 0,Y 177.772,Z 260.784,A -85,B 0,C 180,E1 -23586.812,E2 -23586.812} C_VEL
LIN {X 0,Y 178.979,Z 262.558,A -85,B 0,C 180,E1 -23590.464,E2 -23590.464} C_VEL
LIN {X 0,Y 181.641,Z 265.75,A -85,B 0,C 180,E1 -23595.283,E2 -23595.283} C_VEL
LIN {X 0,Y 185.888,Z 271.489,A -85,B 0,C 180,E1 -23600.528,E2 -23600.528} C_VEL
LIN {X 0,Y 190.111,Z 277.667,A -85,B 0,C 180,E1 -23604.503,E2 -23604.503} C_VEL
LIN {X 0,Y 193.619,Z 282.939,A -85,B 0,C 180,E1 -23607.271,E2 -23607.271} C_VEL
LIN {X 0,Y 196.854,Z 288.16,A -85,B 0,C 180,E1 -23609.547,E2 -23609.547} C_VEL
LIN {X 0,Y 201.001,Z 295.228,A -85,B 0,C 180,E1 -23612.164,E2 -23612.164} C_VEL
LIN {X 0,Y 205.65,Z 304.033,A -85,B 0,C 180,E1 -23614.816,E2 -23614.816} C_VEL
LIN {X 0,Y 210.099,Z 313.233,A -85,B 0,C 180,E1 -23617.13,E2 -23617.13} C_VEL
LIN {X 0,Y 213.91,Z 322.241,A -85,B 0,C 180,E1 -23619.001,E2 -23619.001} C_VEL
LIN {X 0,Y 208.686,Z 394.35,A -85,B 0,C 180,E1 -23621.061,E2 -23621.061} C_VEL
LIN {X 0,Y 206.682,Z 408.723,A -85,B 0,C 180,E1 -23621.758,E2 -23621.758} C_VEL
LIN {X 0,Y 203.97,Z 422.444,A -85,B 0,C 180,E1 -23622.748,E2 -23622.748} C_VEL
LIN {X 0,Y 200.409,Z 435.863,A -85,B 0,C 180,E1 -23624.036,E2 -23624.036} C_VEL
LIN {X 0,Y 196.546,Z 447.724,A -85,B 0,C 180,E1 -23625.505,E2 -23625.505} C_VEL
LIN {X 0,Y 191.718,Z 460.708,A -85,B 0,C 180,E1 -23627.655,E2 -23627.655} C_VEL
LIN {X 0,Y 187.244,Z 470.643,A -85,B 0,C 180,E1 -23629.649,E2 -23629.649} C_VEL
LIN {X 0,Y 181.776,Z 481.659,A -85,B 0,C 180,E1 -23632.486,E2 -23632.486} C_VEL
LIN {X 0,Y 176.743,Z 490.819,A -85,B 0,C 180,E1 -23635.483,E2 -23635.483} C_VEL
LIN {X 0,Y 171.26,Z 499.853,A -85,B 0,C 180,E1 -23639.275,E2 -23639.275} C_VEL
LIN {X 0,Y 167.728,Z 505.874,A -85,B 0,C 180,E1 -23642.553,E2 -23642.553} C_VEL
LIN {X 0,Y 163.028,Z 512.676,A -85,B 0,C 180,E1 -23647.17,E2 -23647.17} C_VEL
LIN {X 0,Y 159.68,Z 517.845,A -85,B 0,C 180,E1 -23652.055,E2 -23652.055} C_VEL
LIN {X 0,Y 157.275,Z 521.596,A -85,B 0,C 180,E1 -23657.089,E2 -23657.089} C_VEL
LIN {X 0,Y 155.857,Z 524.044,A -85,B 0,C 180,E1 -23662.224,E2 -23662.224} C_VEL
LIN {X 0,Y 155.204,Z 525.264,A -85,B 0,C 180,E1 -23667.404,E2 -23667.404} C_VEL
LIN {X 0,Y 155.19,Z 525.282,A -85,B 0,C 180,E1 -23672.595,E2 -23672.595} C_VEL
LIN {X 0,Y 155.794,Z 524.104,A -85,B 0,C 180,E1 -23677.777,E2 -23677.777} C_VEL
LIN {X 0,Y 157.215,Z 521.696,A -85,B 0,C 180,E1 -23682.914,E2 -23682.914} C_VEL
LIN {X 0,Y 159.618,Z 517.984,A -85,B 0,C 180,E1 -23687.95,E2 -23687.95} C_VEL
LIN {X 0,Y 162.971,Z 512.871,A -85,B 0,C 180,E1 -23692.836,E2 -23692.836} C_VEL
LIN {X 0,Y 167.559,Z 506.151,A -85,B 0,C 180,E1 -23697.475,E2 -23697.475} C_VEL
LIN {X 0,Y 172.029,Z 498.801,A -85,B 0,C 180,E1 -23701.39,E2 -23701.39} C_VEL
LIN {X 0,Y 176.648,Z 491.178,A -85,B 0,C 180,E1 -23704.536,E2 -23704.536} C_VEL
LIN {X 0,Y 181.709,Z 482.085,A -85,B 0,C 180,E1 -23707.528,E2 -23707.528} C_VEL
LIN {X 0,Y 187.228,Z 471.162,A -85,B 0,C 180,E1 -23710.353,E2 -23710.353} C_VEL
LIN {X 0,Y 192.129,Z 460.175,A -85,B 0,C 180,E1 -23712.578,E2 -23712.578} C_VEL
LIN {X 0,Y 196.589,Z 448.19,A -85,B 0,C 180,E1 -23714.552,E2 -23714.552} C_VEL
LIN {X 0,Y 200.853,Z 435.032,A -85,B 0,C 180,E1 -23716.192,E2 -23716.192} C_VEL
LIN {X 0,Y 204.107,Z 422.493,A -85,B 0,C 180,E1 -23717.39,E2 -23717.39} C_VEL
LIN {X 0,Y 206.992,Z 408.096,A -85,B 0,C 180,E1 -23718.407,E2 -23718.407} C_VEL
LIN {X 0,Y 208.94,Z 393.695,A -85,B 0,C 180,E1 -23719.098,E2 -23719.098} C_VEL
LIN {X 0,Y 214.108,Z 322.37,A -85,B 0,C 180,E1 -23721.114,E2 -23721.114} C_VEL
LIN {X 0,Y 208.672,Z 309.931,A -85,B 0,C 180,E1 -23723.812,E2 -23723.812} C_VEL
LIN {X 0,Y 203.22,Z 299.144,A -85,B 0,C 180,E1 -23726.775,E2 -23726.775} C_VEL
LIN {X 0,Y 198.092,Z 290.043,A -85,B 0,C 180,E1 -23729.903,E2 -23729.903} C_VEL
LIN {X 0,Y 194.272,Z 283.862,A -85,B 0,C 180,E1 -23732.532,E2 -23732.532} C_VEL
LIN {X 0,Y 191.541,Z 279.785,A -85,B 0,C 180,E1 -23734.616,E2 -23734.616} C_VEL
LIN {X 0,Y 188.696,Z 275.561,A -85,B 0,C 180,E1 -23737.058,E2 -23737.058} C_VEL
LIN {X 0,Y 185.313,Z 270.643,A -85,B 0,C 180,E1 -23740.475,E2 -23740.475} C_VEL
LIN {X 0,Y 181.205,Z 265.041,A -85,B 0,C 180,E1 -23745.957,E2 -23745.957} C_VEL
LIN {X 0,Y 178.235,Z 261.319,A -85,B 0,C 180,E1 -23752.637,E2 -23752.637} C_VEL
LIN {X 0,Y 177.456,Z 259.909,A -85,B 0,C 180,E1 -23758.865,E2 -23758.865} C_VEL
LIN {X 0,Y 177.608,Z 260.117,A -85,B 0,C 180,E1 -23761.133,E2 -23761.133} C_VEL
LIN {X 0,Y 179.102,Z 262.476,A -85,B 0,C 180,E1 -23767.058,E2 -23767.058} C_VEL
LIN {X 0,Y 181.706,Z 265.692,A -85,B 0,C 180,E1 -23771.999,E2 -23771.999} C_VEL
LIN {X 0,Y 186.134,Z 271.806,A -85,B 0,C 180,E1 -23777.581,E2 -23777.581} C_VEL
LIN {X 0,Y 190.316,Z 277.757,A -85,B 0,C 180,E1 -23781.529,E2 -23781.529} C_VEL
LIN {X 0,Y 193.941,Z 283.326,A -85,B 0,C 180,E1 -23784.414,E2 -23784.414} C_VEL
LIN {X 0,Y 197.232,Z 288.607,A -85,B 0,C 180,E1 -23786.735,E2 -23786.735} C_VEL
LIN {X 0,Y 201.526,Z 295.96,A -85,B 0,C 180,E1 -23789.452,E2 -23789.452} C_VEL
LIN {X 0,Y 206.61,Z 305.679,A -85,B 0,C 180,E1 -23792.349,E2 -23792.349} C_VEL
LIN {X 0,Y 212.271,Z 317.793,A -85,B 0,C 180,E1 -23795.267,E2 -23795.267} C_VEL
LIN {X 0,Y 214.26,Z 322.468,A -85,B 0,C 180,E1 -23796.235,E2 -23796.235} C_VEL
LIN {X 0,Y 208.153,Z 401.493,A -85,B 0,C 180,E1 -23798.587,E2 -23798.587} C_VEL
LIN {X 0,Y 205.783,Z 416.853,A -85,B 0,C 180,E1 -23799.309,E2 -23799.309} C_VEL
LIN {X 0,Y 205.177,Z 420.192,A -85,B 0,C 180,E1 -23799.527,E2 -23799.527} C_VEL
LIN {X 0,Y 203.474,Z 425.814,A -85,B 0,C 180,E1 -23799.731,E2 -23799.731} C_VEL
LIN {X 0,Y 199.341,Z 434.823,A -85,B 0,C 180,E1 -23799.838,E2 -23799.838} C_VEL
LIN {X 0,Y 194.908,Z 443.7,A -85,B 0,C 180,E1 -23800.086,E2 -23800.086} C_VEL
LIN {X 0,Y 192.738,Z 448.904,A -85,B 0,C 180,E1 -23800.52,E2 -23800.52} C_VEL
LIN {X 0,Y 187.866,Z 462.212,A -85,B 0,C 180,E1 -23802.328,E2 -23802.328} C_VEL
LIN {X 0,Y 182.453,Z 474.864,A -85,B 0,C 180,E1 -23804.554,E2 -23804.554} C_VEL
LIN {X 0,Y 177.322,Z 485.29,A -85,B 0,C 180,E1 -23806.869,E2 -23806.869} C_VEL
LIN {X 0,Y 171.644,Z 495.871,A -85,B 0,C 180,E1 -23809.845,E2 -23809.845} C_VEL
LIN {X 0,Y 166.554,Z 504.771,A -85,B 0,C 180,E1 -23813.039,E2 -23813.039} C_VEL
LIN {X 0,Y 161.437,Z 513.482,A -85,B 0,C 180,E1 -23817.033,E2 -23817.033} C_VEL
LIN {X 0,Y 156.325,Z 521.575,A -85,B 0,C 180,E1 -23821.834,E2 -23821.834} C_VEL
LIN {X 0,Y 152.415,Z 528.052,A -85,B 0,C 180,E1 -23827.002,E2 -23827.002} C_VEL
LIN {X 0,Y 149.776,Z 532.871,A -85,B 0,C 180,E1 -23832.243,E2 -23832.243} C_VEL
LIN {X 0,Y 148.461,Z 535.629,A -85,B 0,C 180,E1 -23836.31,E2 -23836.31} C_VEL
LIN {X 0,Y 147.754,Z 538.186,A -85,B 0,C 180,E1 -23841.797,E2 -23841.797} C_VEL
LIN {X 0,Y 147.823,Z 539.477,A -85,B 0,C 180,E1 -23847.276,E2 -23847.276} C_VEL
LIN {X 0,Y 147.967,Z 539.644,A -85,B 0,C 180,E1 -23850.001,E2 -23850.001} C_VEL
LIN {X 0,Y 147.818,Z 539.398,A -85,B 0,C 180,E1 -23853.201,E2 -23853.201} C_VEL
LIN {X 0,Y 147.757,Z 538.156,A -85,B 0,C 180,E1 -23858.205,E2 -23858.205} C_VEL
LIN {X 0,Y 148.477,Z 535.578,A -85,B 0,C 180,E1 -23863.691,E2 -23863.691} C_VEL
LIN {X 0,Y 150.351,Z 531.698,A -85,B 0,C 180,E1 -23869.1,E2 -23869.1} C_VEL
LIN {X 0,Y 153.333,Z 526.415,A -85,B 0,C 180,E1 -23874.364,E2 -23874.364} C_VEL
LIN {X 0,Y 157.457,Z 519.593,A -85,B 0,C 180,E1 -23879.405,E2 -23879.405} C_VEL
LIN {X 0,Y 162.093,Z 512.183,A -85,B 0,C 180,E1 -23883.561,E2 -23883.561} C_VEL
LIN {X 0,Y 167.328,Z 503.205,A -85,B 0,C 180,E1 -23887.519,E2 -23887.519} C_VEL
LIN {X 0,Y 172.538,Z 493.993,A -85,B 0,C 180,E1 -23890.672,E2 -23890.672} C_VEL
LIN {X 0,Y 178.241,Z 483.042,A -85,B 0,C 180,E1 -23893.632,E2 -23893.632} C_VEL
LIN {X 0,Y 184.028,Z 470.993,A -85,B 0,C 180,E1 -23896.124,E2 -23896.124} C_VEL
LIN {X 0,Y 188.866,Z 459.09,A -85,B 0,C 180,E1 -23898.093,E2 -23898.093} C_VEL
LIN {X 0,Y 193.399,Z 446.252,A -85,B 0,C 180,E1 -23899.741,E2 -23899.741} C_VEL
LIN {X 0,Y 197.546,Z 432.191,A -85,B 0,C 180,E1 -23901.1,E2 -23901.1} C_VEL
LIN {X 0,Y 200.867,Z 417.653,A -85,B 0,C 180,E1 -23902.132,E2 -23902.132} C_VEL
LIN {X 0,Y 203.133,Z 404.051,A -85,B 0,C 180,E1 -23902.799,E2 -23902.799} C_VEL
LIN {X 0,Y 204.874,Z 385.094,A -85,B 0,C 180,E1 -23903.45,E2 -23903.45} C_VEL
LIN {X 0,Y 209.637,Z 325.03,A -85,B 0,C 180,E1 -23905.176,E2 -23905.176} C_VEL
LIN {X 0,Y 205.147,Z 314.742,A -85,B 0,C 180,E1 -23907.564,E2 -23907.564} C_VEL
LIN {X 0,Y 200.196,Z 304.468,A -85,B 0,C 180,E1 -23910.45,E2 -23910.45} C_VEL
LIN {X 0,Y 195.815,Z 296.41,A -85,B 0,C 180,E1 -23913.272,E2 -23913.272} C_VEL
LIN {X 0,Y 192.426,Z 290.672,A -85,B 0,C 180,E1 -23915.704,E2 -23915.704} C_VEL
LIN {X 0,Y 189.835,Z 286.573,A -85,B 0,C 180,E1 -23917.756,E2 -23917.756} C_VEL
LIN {X 0,Y 186.92,Z 281.973,A -85,B 0,C 180,E1 -23920.365,E2 -23920.365} C_VEL
LIN {X 0,Y 183.688,Z 277.236,A -85,B 0,C 180,E1 -23923.748,E2 -23923.748} C_VEL
LIN {X 0,Y 179.871,Z 271.775,A -85,B 0,C 180,E1 -23929.02,E2 -23929.02} C_VEL
LIN {X 0,Y 177.15,Z 268.148,A -85,B 0,C 180,E1 -23935.202,E2 -23935.202} C_VEL
LIN {X 0,Y 176.344,Z 266.62,A -85,B 0,C 180,E1 -23940,E2 -23940} C_VEL
LIN {X 0,Y 176.81,Z 267.713,A -85,B 0,C 180,E1 -23946.423,E2 -23946.423} C_VEL
LIN {X 0,Y 177.885,Z 269.407,A -85,B 0,C 180,E1 -23949.954,E2 -23949.954} C_VEL
LIN {X 0,Y 180.34,Z 272.451,A -85,B 0,C 180,E1 -23954.674,E2 -23954.674} C_VEL
LIN {X 0,Y 184.361,Z 278.181,A -85,B 0,C 180,E1 -23959.92,E2 -23959.92} C_VEL
LIN {X 0,Y 188.196,Z 283.998,A -85,B 0,C 180,E1 -23963.72,E2 -23963.72} C_VEL
LIN {X 0,Y 191.677,Z 289.431,A -85,B 0,C 180,E1 -23966.604,E2 -23966.604} C_VEL
LIN {X 0,Y 195.175,Z 295.343,A -85,B 0,C 180,E1 -23969.16,E2 -23969.16} C_VEL
LIN {X 0,Y 199.579,Z 303.406,A -85,B 0,C 180,E1 -23972.028,E2 -23972.028} C_VEL
LIN {X 0,Y 203.924,Z 312.055,A -85,B 0,C 180,E1 -23974.572,E2 -23974.572} C_VEL
LIN {X 0,Y 208.81,Z 323.254,A -85,B 0,C 180,E1 -23977.204,E2 -23977.204} C_VEL
LIN {X 0,Y 209.436,Z 324.812,A -85,B 0,C 180,E1 -23977.527,E2 -23977.527} C_VEL
LIN {X 0,Y 204.515,Z 391.288,A -85,B 0,C 180,E1 -23979.42,E2 -23979.42} C_VEL
LIN {X 0,Y 202.694,Z 405.615,A -85,B 0,C 180,E1 -23980.054,E2 -23980.054} C_VEL
LIN {X 0,Y 200.073,Z 419.292,A -85,B 0,C 180,E1 -23980.954,E2 -23980.954} C_VEL
LIN {X 0,Y 196.687,Z 432.545,A -85,B 0,C 180,E1 -23982.146,E2 -23982.146} C_VEL
LIN {X 0,Y 192.183,Z 446.316,A -85,B 0,C 180,E1 -23983.76,E2 -23983.76} C_VEL
LIN {X 0,Y 187.601,Z 458.674,A -85,B 0,C 180,E1 -23985.754,E2 -23985.754} C_VEL
LIN {X 0,Y 182.449,Z 469.969,A -85,B 0,C 180,E1 -23987.987,E2 -23987.987} C_VEL
LIN {X 0,Y 177.139,Z 480.305,A -85,B 0,C 180,E1 -23990.594,E2 -23990.594} C_VEL
LIN {X 0,Y 171.826,Z 489.722,A -85,B 0,C 180,E1 -23993.624,E2 -23993.624} C_VEL
LIN {X 0,Y 166.836,Z 497.613,A -85,B 0,C 180,E1 -23996.795,E2 -23996.795} C_VEL
LIN {X 0,Y 163.095,Z 503.49,A -85,B 0,C 180,E1 -23999.743,E2 -23999.743} C_VEL
LIN {X 0,Y 160.142,Z 508.053,A -85,B 0,C 180,E1 -24002.56,E2 -24002.56} C_VEL
LIN {X 0,Y 155.493,Z 514.412,A -85,B 0,C 180,E1 -24007.406,E2 -24007.406} C_VEL
LIN {X 0,Y 152.174,Z 519.216,A -85,B 0,C 180,E1 -24012.53,E2 -24012.53} C_VEL
LIN {X 0,Y 150.358,Z 521.93,A -85,B 0,C 180,E1 -24016.484,E2 -24016.484} C_VEL
LIN {X 0,Y 148.835,Z 524.377,A -85,B 0,C 180,E1 -24021.855,E2 -24021.855} C_VEL
LIN {X 0,Y 148.119,Z 525.597,A -85,B 0,C 180,E1 -24027.279,E2 -24027.279} C_VEL
LIN {X 0,Y 148.104,Z 525.615,A -85,B 0,C 180,E1 -24032.719,E2 -24032.719} C_VEL
LIN {X 0,Y 148.764,Z 524.437,A -85,B 0,C 180,E1 -24038.147,E2 -24038.147} C_VEL
LIN {X 0,Y 150.306,Z 522.029,A -85,B 0,C 180,E1 -24043.519,E2 -24043.519} C_VEL
LIN {X 0,Y 152.861,Z 518.318,A -85,B 0,C 180,E1 -24048.773,E2 -24048.773} C_VEL
LIN {X 0,Y 156.46,Z 513.205,A -85,B 0,C 180,E1 -24053.844,E2 -24053.844} C_VEL
LIN {X 0,Y 160.03,Z 508.296,A -85,B 0,C 180,E1 -24057.458,E2 -24057.458} C_VEL
LIN {X 0,Y 164.528,Z 501.37,A -85,B 0,C 180,E1 -24061.55,E2 -24061.55} C_VEL
LIN {X 0,Y 169.978,Z 492.86,A -85,B 0,C 180,E1 -24065.368,E2 -24065.368} C_VEL
LIN {X 0,Y 175.231,Z 484.046,A -85,B 0,C 180,E1 -24068.436,E2 -24068.436} C_VEL
LIN {X 0,Y 180.852,Z 473.465,A -85,B 0,C 180,E1 -24071.346,E2 -24071.346} C_VEL
LIN {X 0,Y 185.899,Z 462.97,A -85,B 0,C 180,E1 -24073.59,E2 -24073.59} C_VEL
LIN {X 0,Y 190.858,Z 450.582,A -85,B 0,C 180,E1 -24075.741,E2 -24075.741} C_VEL
LIN {X 0,Y 194.901,Z 439.009,A -85,B 0,C 180,E1 -24077.281,E2 -24077.281} C_VEL
LIN {X 0,Y 198.81,Z 425.275,A -85,B 0,C 180,E1 -24078.692,E2 -24078.692} C_VEL
LIN {X 0,Y 201.957,Z 410.942,A -85,B 0,C 180,E1 -24079.764,E2 -24079.764} C_VEL
LIN {X 0,Y 204.2,Z 396.042,A -85,B 0,C 180,E1 -24080.536,E2 -24080.536} C_VEL
LIN {X 0,Y 206.301,Z 370.951,A -85,B 0,C 180,E1 -24081.289,E2 -24081.289} C_VEL
LIN {X 0,Y 209.61,Z 324.903,A -85,B 0,C 180,E1 -24082.604,E2 -24082.604} C_VEL
LIN {X 0,Y 204.553,Z 313.22,A -85,B 0,C 180,E1 -24085.306,E2 -24085.306} C_VEL
LIN {X 0,Y 199.842,Z 303.755,A -85,B 0,C 180,E1 -24088.055,E2 -24088.055} C_VEL
LIN {X 0,Y 195.372,Z 295.543,A -85,B 0,C 180,E1 -24090.973,E2 -24090.973} C_VEL
LIN {X 0,Y 191.995,Z 289.868,A -85,B 0,C 180,E1 -24093.442,E2 -24093.442} C_VEL
LIN {X 0,Y 189.613,Z 286.128,A -85,B 0,C 180,E1 -24095.363,E2 -24095.363} C_VEL
LIN {X 0,Y 186.68,Z 281.644,A -85,B 0,C 180,E1 -24098.031,E2 -24098.031} C_VEL
LIN {X 0,Y 183.753,Z 277.226,A -85,B 0,C 180,E1 -24101.173,E2 -24101.173} C_VEL
LIN {X 0,Y 180.005,Z 271.893,A -85,B 0,C 180,E1 -24106.452,E2 -24106.452} C_VEL
LIN {X 0,Y 177.223,Z 268.216,A -85,B 0,C 180,E1 -24113.167,E2 -24113.167} C_VEL
LIN {X 0,Y 176.59,Z 267.101,A -85,B 0,C 180,E1 -24117.719,E2 -24117.719} C_VEL
LIN {X 0,Y 176.687,Z 267.042,A -85,B 0,C 180,E1 -24120.569,E2 -24120.569} C_VEL
LIN {X 0,Y 178.115,Z 269.442,A -85,B 0,C 180,E1 -24126.798,E2 -24126.798} C_VEL
LIN {X 0,Y 180.479,Z 272.532,A -85,B 0,C 180,E1 -24131.512,E2 -24131.512} C_VEL
LIN {X 0,Y 184.589,Z 278.441,A -85,B 0,C 180,E1 -24136.962,E2 -24136.962} C_VEL
LIN {X 0,Y 188.329,Z 284.002,A -85,B 0,C 180,E1 -24140.692,E2 -24140.692} C_VEL
LIN {X 0,Y 192.038,Z 289.918,A -85,B 0,C 180,E1 -24143.796,E2 -24143.796} C_VEL
LIN {X 0,Y 196.292,Z 297.04,A -85,B 0,C 180,E1 -24146.873,E2 -24146.873} C_VEL
LIN {X 0,Y 201.179,Z 306.271,A -85,B 0,C 180,E1 -24149.999,E2 -24149.999} C_VEL
LIN {X 0,Y 206.169,Z 316.751,A -85,B 0,C 180,E1 -24152.857,E2 -24152.857} C_VEL
LIN {X 0,Y 209.812,Z 325.247,A -85,B 0,C 180,E1 -24154.791,E2 -24154.791} C_VEL
LIN {X 0,Y 203.719,Z 401.129,A -85,B 0,C 180,E1 -24157.042,E2 -24157.042} C_VEL
LIN {X 0,Y 201.36,Z 416.215,A -85,B 0,C 180,E1 -24157.746,E2 -24157.746} C_VEL
LIN {X 0,Y 198.172,Z 430.559,A -85,B 0,C 180,E1 -24158.722,E2 -24158.722} C_VEL
LIN {X 0,Y 194.02,Z 444.984,A -85,B 0,C 180,E1 -24160.076,E2 -24160.076} C_VEL
LIN {X 0,Y 192.738,Z 448.904,A -85,B 0,C 180,E1 -24160.52,E2 -24160.52} C_VEL
LIN {X 0,Y 190.452,Z 454.119,A -85,B 0,C 180,E1 -24161.005,E2 -24161.005} C_VEL
LIN {X 0,Y 185.31,Z 462.419,A -85,B 0,C 180,E1 -24161.556,E2 -24161.556} C_VEL
LIN {X 0,Y 179.898,Z 470.389,A -85,B 0,C 180,E1 -24162.275,E2 -24162.275} C_VEL
LIN {X 0,Y 177.219,Z 475.084,A -85,B 0,C 180,E1 -24163.036,E2 -24163.036} C_VEL
LIN {X 0,Y 171.135,Z 486.842,A -85,B 0,C 180,E1 -24165.724,E2 -24165.724} C_VEL
LIN {X 0,Y 165.296,Z 497.132,A -85,B 0,C 180,E1 -24168.776,E2 -24168.776} C_VEL
LIN {X 0,Y 159.345,Z 506.916,A -85,B 0,C 180,E1 -24172.551,E2 -24172.551} C_VEL
LIN {X 0,Y 154.015,Z 515.355,A -85,B 0,C 180,E1 -24176.8,E2 -24176.8} C_VEL
LIN {X 0,Y 150.016,Z 521.233,A -85,B 0,C 180,E1 -24180.536,E2 -24180.536} C_VEL
LIN {X 0,Y 145.78,Z 527.78,A -85,B 0,C 180,E1 -24185.962,E2 -24185.962} C_VEL
LIN {X 0,Y 142.949,Z 532.533,A -85,B 0,C 180,E1 -24191.365,E2 -24191.365} C_VEL
LIN {X 0,Y 141.497,Z 535.293,A -85,B 0,C 180,E1 -24195.622,E2 -24195.622} C_VEL
LIN {X 0,Y 140.674,Z 537.851,A -85,B 0,C 180,E1 -24201.381,E2 -24201.381} C_VEL
LIN {X 0,Y 140.734,Z 539.144,A -85,B 0,C 180,E1 -24207.139,E2 -24207.139} C_VEL
LIN {X 0,Y 140.874,Z 539.311,A -85,B 0,C 180,E1 -24210.001,E2 -24210.001} C_VEL
LIN {X 0,Y 140.735,Z 539.137,A -85,B 0,C 180,E1 -24212.863,E2 -24212.863} C_VEL
LIN {X 0,Y 140.677,Z 537.82,A -85,B 0,C 180,E1 -24218.621,E2 -24218.621} C_VEL
LIN {X 0,Y 141.515,Z 535.24,A -85,B 0,C 180,E1 -24224.379,E2 -24224.379} C_VEL
LIN {X 0,Y 143.588,Z 531.359,A -85,B 0,C 180,E1 -24230.037,E2 -24230.037} C_VEL
LIN {X 0,Y 146.8,Z 526.073,A -85,B 0,C 180,E1 -24235.524,E2 -24235.524} C_VEL
LIN {X 0,Y 151.242,Z 519.248,A -85,B 0,C 180,E1 -24240.741,E2 -24240.741} C_VEL
LIN {X 0,Y 156.124,Z 511.831,A -85,B 0,C 180,E1 -24245.026,E2 -24245.026} C_VEL
LIN {X 0,Y 161.687,Z 502.849,A -85,B 0,C 180,E1 -24249.07,E2 -24249.07} C_VEL
LIN {X 0,Y 167.16,Z 493.627,A -85,B 0,C 180,E1 -24252.276,E2 -24252.276} C_VEL
LIN {X 0,Y 173.151,Z 482.664,A -85,B 0,C 180,E1 -24255.26,E2 -24255.26} C_VEL
LIN {X 0,Y 179.148,Z 470.594,A -85,B 0,C 180,E1 -24257.772,E2 -24257.772} C_VEL
LIN {X 0,Y 184.169,Z 458.661,A -85,B 0,C 180,E1 -24259.749,E2 -24259.749} C_VEL
LIN {X 0,Y 188.882,Z 445.781,A -85,B 0,C 180,E1 -24261.387,E2 -24261.387} C_VEL
LIN {X 0,Y 193.107,Z 431.644,A -85,B 0,C 180,E1 -24262.762,E2 -24262.762} C_VEL
LIN {X 0,Y 196.278,Z 418.517,A -85,B 0,C 180,E1 -24263.673,E2 -24263.673} C_VEL
LIN {X 0,Y 198.785,Z 403.952,A -85,B 0,C 180,E1 -24264.406,E2 -24264.406} C_VEL
LIN {X 0,Y 200.586,Z 385.16,A -85,B 0,C 180,E1 -24265.051,E2 -24265.051} C_VEL
LIN {X 0,Y 205.261,Z 327.761,A -85,B 0,C 180,E1 -24266.709,E2 -24266.709} C_VEL
LIN {X 0,Y 201.223,Z 318.305,A -85,B 0,C 180,E1 -24269.031,E2 -24269.031} C_VEL
LIN {X 0,Y 196.861,Z 309.038,A -85,B 0,C 180,E1 -24271.769,E2 -24271.769} C_VEL
LIN {X 0,Y 192.742,Z 301.203,A -85,B 0,C 180,E1 -24274.632,E2 -24274.632} C_VEL
LIN {X 0,Y 189.578,Z 295.686,A -85,B 0,C 180,E1 -24277.092,E2 -24277.092} C_VEL
LIN {X 0,Y 187.208,Z 291.822,A -85,B 0,C 180,E1 -24279.132,E2 -24279.132} C_VEL
LIN {X 0,Y 184.959,Z 288.156,A -85,B 0,C 180,E1 -24281.301,E2 -24281.301} C_VEL
LIN {X 0,Y 182.115,Z 283.789,A -85,B 0,C 180,E1 -24284.471,E2 -24284.471} C_VEL
LIN {X 0,Y 178.674,Z 278.585,A -85,B 0,C 180,E1 -24289.519,E2 -24289.519} C_VEL
LIN {X 0,Y 176.21,Z 275.161,A -85,B 0,C 180,E1 -24295.425,E2 -24295.425} C_VEL
LIN {X 0,Y 175.479,Z 273.667,A -85,B 0,C 180,E1 -24300,E2 -24300} C_VEL
LIN {X 0,Y 175.947,Z 274.789,A -85,B 0,C 180,E1 -24306.455,E2 -24306.455} C_VEL
LIN {X 0,Y 178.045,Z 277.92,A -85,B 0,C 180,E1 -24312.25,E2 -24312.25} C_VEL
LIN {X 0,Y 179.213,Z 279.487,A -85,B 0,C 180,E1 -24314.333,E2 -24314.333} C_VEL
LIN {X 0,Y 182.845,Z 284.841,A -85,B 0,C 180,E1 -24319.289,E2 -24319.289} C_VEL
LIN {X 0,Y 186.306,Z 290.307,A -85,B 0,C 180,E1 -24322.908,E2 -24322.908} C_VEL
LIN {X 0,Y 189.782,Z 295.992,A -85,B 0,C 180,E1 -24325.941,E2 -24325.941} C_VEL
LIN {X 0,Y 193.501,Z 302.559,A -85,B 0,C 180,E1 -24328.767,E2 -24328.767} C_VEL
LIN {X 0,Y 198.077,Z 311.502,A -85,B 0,C 180,E1 -24331.845,E2 -24331.845} C_VEL
LIN {X 0,Y 202.152,Z 320.353,A -85,B 0,C 180,E1 -24334.318,E2 -24334.318} C_VEL
LIN {X 0,Y 205.11,Z 327.517,A -85,B 0,C 180,E1 -24335.998,E2 -24335.998} C_VEL
LIN {X 0,Y 200.738,Z 385.669,A -85,B 0,C 180,E1 -24337.653,E2 -24337.653} C_VEL
LIN {X 0,Y 199.133,Z 400.548,A -85,B 0,C 180,E1 -24338.189,E2 -24338.189} C_VEL
LIN {X 0,Y 196.671,Z 414.624,A -85,B 0,C 180,E1 -24338.992,E2 -24338.992} C_VEL
LIN {X 0,Y 193.183,Z 429.085,A -85,B 0,C 180,E1 -24340.183,E2 -24340.183} C_VEL
LIN {X 0,Y 189.109,Z 442.031,A -85,B 0,C 180,E1 -24341.589,E2 -24341.589} C_VEL
LIN {X 0,Y 184.681,Z 453.909,A -85,B 0,C 180,E1 -24343.287,E2 -24343.287} C_VEL
LIN {X 0,Y 179.405,Z 466.115,A -85,B 0,C 180,E1 -24345.554,E2 -24345.554} C_VEL
LIN {X 0,Y 173.687,Z 477.152,A -85,B 0,C 180,E1 -24348.114,E2 -24348.114} C_VEL
LIN {X 0,Y 167.989,Z 487.149,A -85,B 0,C 180,E1 -24351.131,E2 -24351.131} C_VEL
LIN {X 0,Y 162.612,Z 495.523,A -85,B 0,C 180,E1 -24354.305,E2 -24354.305} C_VEL
LIN {X 0,Y 157.428,Z 503.113,A -85,B 0,C 180,E1 -24358.019,E2 -24358.019} C_VEL
LIN {X 0,Y 153.884,Z 508.392,A -85,B 0,C 180,E1 -24361.344,E2 -24361.344} C_VEL
LIN {X 0,Y 148.964,Z 514.748,A -85,B 0,C 180,E1 -24366.357,E2 -24366.357} C_VEL
LIN {X 0,Y 145.404,Z 519.551,A -85,B 0,C 180,E1 -24371.688,E2 -24371.688} C_VEL
LIN {X 0,Y 143.47,Z 522.263,A -85,B 0,C 180,E1 -24375.821,E2 -24375.821} C_VEL
LIN {X 0,Y 141.811,Z 524.711,A -85,B 0,C 180,E1 -24381.449,E2 -24381.449} C_VEL
LIN {X 0,Y 141.037,Z 525.93,A -85,B 0,C 180,E1 -24387.143,E2 -24387.143} C_VEL
LIN {X 0,Y 141.021,Z 525.947,A -85,B 0,C 180,E1 -24392.856,E2 -24392.856} C_VEL
LIN {X 0,Y 141.735,Z 524.77,A -85,B 0,C 180,E1 -24398.554,E2 -24398.554} C_VEL
LIN {X 0,Y 143.398,Z 522.362,A -85,B 0,C 180,E1 -24404.184,E2 -24404.184} C_VEL
LIN {X 0,Y 146.147,Z 518.651,A -85,B 0,C 180,E1 -24409.67,E2 -24409.67} C_VEL
LIN {X 0,Y 150.005,Z 513.538,A -85,B 0,C 180,E1 -24414.938,E2 -24414.938} C_VEL
LIN {X 0,Y 153.759,Z 508.634,A -85,B 0,C 180,E1 -24418.679,E2 -24418.679} C_VEL
LIN {X 0,Y 158.525,Z 501.711,A -85,B 0,C 180,E1 -24422.892,E2 -24422.892} C_VEL
LIN {X 0,Y 164.257,Z 493.206,A -85,B 0,C 180,E1 -24426.798,E2 -24426.798} C_VEL
LIN {X 0,Y 169.727,Z 484.402,A -85,B 0,C 180,E1 -24429.926,E2 -24429.926} C_VEL
LIN {X 0,Y 175.605,Z 473.833,A -85,B 0,C 180,E1 -24432.871,E2 -24432.871} C_VEL
LIN {X 0,Y 181.299,Z 462.409,A -85,B 0,C 180,E1 -24435.31,E2 -24435.31} C_VEL
LIN {X 0,Y 186.208,Z 450.437,A -85,B 0,C 180,E1 -24437.387,E2 -24437.387} C_VEL
LIN {X 0,Y 190.74,Z 437.709,A -85,B 0,C 180,E1 -24439.053,E2 -24439.053} C_VEL
LIN {X 0,Y 194.523,Z 424.67,A -85,B 0,C 180,E1 -24440.352,E2 -24440.352} C_VEL
LIN {X 0,Y 197.768,Z 410.055,A -85,B 0,C 180,E1 -24441.424,E2 -24441.424} C_VEL
LIN {X 0,Y 199.978,Z 395.429,A -85,B 0,C 180,E1 -24442.162,E2 -24442.162} C_VEL
LIN {X 0,Y 202.828,Z 361.141,A -85,B 0,C 180,E1 -24443.156,E2 -24443.156} C_VEL
LIN {X 0,Y 205.33,Z 327.679,A -85,B 0,C 180,E1 -24444.115,E2 -24444.115} C_VEL
LIN {X 0,Y 200.668,Z 316.722,A -85,B 0,C 180,E1 -24446.804,E2 -24446.804} C_VEL
LIN {X 0,Y 195.256,Z 305.66,A -85,B 0,C 180,E1 -24450.273,E2 -24450.273} C_VEL
LIN {X 0,Y 190.929,Z 297.737,A -85,B 0,C 180,E1 -24453.451,E2 -24453.451} C_VEL
LIN {X 0,Y 187.651,Z 292.385,A -85,B 0,C 180,E1 -24456.185,E2 -24456.185} C_VEL
LIN {X 0,Y 184.894,Z 287.996,A -85,B 0,C 180,E1 -24458.84,E2 -24458.84} C_VEL
LIN {X 0,Y 182.219,Z 283.808,A -85,B 0,C 180,E1 -24461.882,E2 -24461.882} C_VEL
LIN {X 0,Y 178.777,Z 278.698,A -85,B 0,C 180,E1 -24467.026,E2 -24467.026} C_VEL
LIN {X 0,Y 176.295,Z 275.217,A -85,B 0,C 180,E1 -24473.402,E2 -24473.402} C_VEL
LIN {X 0,Y 175.725,Z 274.028,A -85,B 0,C 180,E1 -24478.945,E2 -24478.945} C_VEL
LIN {X 0,Y 175.874,Z 274.238,A -85,B 0,C 180,E1 -24481.144,E2 -24481.144} C_VEL
LIN {X 0,Y 177.237,Z 276.601,A -85,B 0,C 180,E1 -24486.832,E2 -24486.832} C_VEL
LIN {X 0,Y 179.266,Z 279.363,A -85,B 0,C 180,E1 -24491.018,E2 -24491.018} C_VEL
LIN {X 0,Y 183.068,Z 285.146,A -85,B 0,C 180,E1 -24496.343,E2 -24496.343} C_VEL
LIN {X 0,Y 186.45,Z 290.38,A -85,B 0,C 180,E1 -24499.907,E2 -24499.907} C_VEL
LIN {X 0,Y 189.757,Z 295.842,A -85,B 0,C 180,E1 -24502.84,E2 -24502.84} C_VEL
LIN {X 0,Y 193.374,Z 302.179,A -85,B 0,C 180,E1 -24505.64,E2 -24505.64} C_VEL
LIN {X 0,Y 197.906,Z 310.917,A -85,B 0,C 180,E1 -24508.745,E2 -24508.745} C_VEL
LIN {X 0,Y 202.642,Z 321.247,A -85,B 0,C 180,E1 -24511.655,E2 -24511.655} C_VEL
LIN {X 0,Y 205.447,Z 327.922,A -85,B 0,C 180,E1 -24513.257,E2 -24513.257} C_VEL
LIN {X 0,Y 199.452,Z 400.769,A -85,B 0,C 180,E1 -24515.434,E2 -24515.434} C_VEL
LIN {X 0,Y 197.063,Z 415.572,A -85,B 0,C 180,E1 -24516.101,E2 -24516.101} C_VEL
LIN {X 0,Y 193.788,Z 430.031,A -85,B 0,C 180,E1 -24517.076,E2 -24517.076} C_VEL
LIN {X 0,Y 189.521,Z 444.525,A -85,B 0,C 180,E1 -24518.431,E2 -24518.431} C_VEL
LIN {X 0,Y 184.78,Z 457.636,A -85,B 0,C 180,E1 -24520.056,E2 -24520.056} C_VEL
LIN {X 0,Y 179.704,Z 469.736,A -85,B 0,C 180,E1 -24522.009,E2 -24522.009} C_VEL
LIN {X 0,Y 177.219,Z 475.084,A -85,B 0,C 180,E1 -24523.036,E2 -24523.036} C_VEL
LIN {X 0,Y 174.453,Z 479.676,A -85,B 0,C 180,E1 -24523.857,E2 -24523.857} C_VEL
LIN {X 0,Y 168.487,Z 486.909,A -85,B 0,C 180,E1 -24524.942,E2 -24524.942} C_VEL
LIN {X 0,Y 162.361,Z 493.735,A -85,B 0,C 180,E1 -24526.236,E2 -24526.236} C_VEL
LIN {X 0,Y 159.398,Z 497.66,A -85,B 0,C 180,E1 -24527.396,E2 -24527.396} C_VEL
LIN {X 0,Y 153.321,Z 507.141,A -85,B 0,C 180,E1 -24531.191,E2 -24531.191} C_VEL
LIN {X 0,Y 148.055,Z 515.012,A -85,B 0,C 180,E1 -24535.278,E2 -24535.278} C_VEL
LIN {X 0,Y 143.808,Z 520.891,A -85,B 0,C 180,E1 -24539.128,E2 -24539.128} C_VEL
LIN {X 0,Y 139.337,Z 527.294,A -85,B 0,C 180,E1 -24544.615,E2 -24544.615} C_VEL
LIN {X 0,Y 136.153,Z 532.195,A -85,B 0,C 180,E1 -24550.397,E2 -24550.397} C_VEL
LIN {X 0,Y 134.556,Z 534.956,A -85,B 0,C 180,E1 -24554.863,E2 -24554.863} C_VEL
LIN {X 0,Y 133.595,Z 537.515,A -85,B 0,C 180,E1 -24560.921,E2 -24560.921} C_VEL
LIN {X 0,Y 133.634,Z 538.811,A -85,B 0,C 180,E1 -24566.987,E2 -24566.987} C_VEL
LIN {X 0,Y 133.782,Z 538.979,A -85,B 0,C 180,E1 -24570.001,E2 -24570.001} C_VEL
LIN {X 0,Y 133.634,Z 538.803,A -85,B 0,C 180,E1 -24573.016,E2 -24573.016} C_VEL
LIN {X 0,Y 133.623,Z 537.485,A -85,B 0,C 180,E1 -24579.079,E2 -24579.079} C_VEL
LIN {X 0,Y 134.575,Z 534.903,A -85,B 0,C 180,E1 -24585.137,E2 -24585.137} C_VEL
LIN {X 0,Y 136.863,Z 531.02,A -85,B 0,C 180,E1 -24591.067,E2 -24591.067} C_VEL
LIN {X 0,Y 140.343,Z 525.731,A -85,B 0,C 180,E1 -24596.789,E2 -24596.789} C_VEL
LIN {X 0,Y 145.116,Z 518.905,A -85,B 0,C 180,E1 -24602.191,E2 -24602.191} C_VEL
LIN {X 0,Y 150.301,Z 511.483,A -85,B 0,C 180,E1 -24606.598,E2 -24606.598} C_VEL
LIN {X 0,Y 156.177,Z 502.494,A -85,B 0,C 180,E1 -24610.731,E2 -24610.731} C_VEL
LIN {X 0,Y 161.939,Z 493.263,A -85,B 0,C 180,E1 -24613.979,E2 -24613.979} C_VEL
LIN {X 0,Y 167.095,Z 484.257,A -85,B 0,C 180,E1 -24616.514,E2 -24616.514} C_VEL
LIN {X 0,Y 173.261,Z 472.561,A -85,B 0,C 180,E1 -24619.068,E2 -24619.068} C_VEL
LIN {X 0,Y 179.185,Z 459.316,A -85,B 0,C 180,E1 -24621.329,E2 -24621.329} C_VEL
LIN {X 0,Y 184.519,Z 445.309,A -85,B 0,C 180,E1 -24623.116,E2 -24623.116} C_VEL
LIN {X 0,Y 188.891,Z 431.105,A -85,B 0,C 180,E1 -24624.479,E2 -24624.479} C_VEL
LIN {X 0,Y 192.295,Z 417.095,A -85,B 0,C 180,E1 -24625.434,E2 -24625.434} C_VEL
LIN {X 0,Y 194.72,Z 403.056,A -85,B 0,C 180,E1 -24626.113,E2 -24626.113} C_VEL
LIN {X 0,Y 196.523,Z 384.53,A -85,B 0,C 180,E1 -24626.737,E2 -24626.737} C_VEL
LIN {X 0,Y 201.054,Z 330.441,A -85,B 0,C 180,E1 -24628.304,E2 -24628.304} C_VEL
LIN {X 0,Y 196.203,Z 318.999,A -85,B 0,C 180,E1 -24631.374,E2 -24631.374} C_VEL
LIN {X 0,Y 191.769,Z 309.836,A -85,B 0,C 180,E1 -24634.494,E2 -24634.494} C_VEL
LIN {X 0,Y 188.115,Z 302.958,A -85,B 0,C 180,E1 -24637.412,E2 -24637.412} C_VEL
LIN {X 0,Y 185.569,Z 298.592,A -85,B 0,C 180,E1 -24639.688,E2 -24639.688} C_VEL
LIN {X 0,Y 183.297,Z 294.689,A -85,B 0,C 180,E1 -24641.993,E2 -24641.993} C_VEL
LIN {X 0,Y 180.476,Z 290.193,A -85,B 0,C 180,E1 -24645.338,E2 -24645.338} C_VEL
LIN {X 0,Y 177.497,Z 285.387,A -85,B 0,C 180,E1 -24650.025,E2 -24650.025} C_VEL
LIN {X 0,Y 175.192,Z 282.046,A -85,B 0,C 180,E1 -24655.975,E2 -24655.975} C_VEL
LIN {X 0,Y 174.611,Z 280.733,A -85,B 0,C 180,E1 -24660,E2 -24660} C_VEL
LIN {X 0,Y 175.049,Z 281.836,A -85,B 0,C 180,E1 -24666.339,E2 -24666.339} C_VEL
LIN {X 0,Y 177.189,Z 285.122,A -85,B 0,C 180,E1 -24672.31,E2 -24672.31} C_VEL
LIN {X 0,Y 178.017,Z 286.364,A -85,B 0,C 180,E1 -24673.848,E2 -24673.848} C_VEL
LIN {X 0,Y 181.243,Z 291.306,A -85,B 0,C 180,E1 -24678.511,E2 -24678.511} C_VEL
LIN {X 0,Y 184.479,Z 296.672,A -85,B 0,C 180,E1 -24682.104,E2 -24682.104} C_VEL
LIN {X 0,Y 187.743,Z 302.231,A -85,B 0,C 180,E1 -24685.116,E2 -24685.116} C_VEL
LIN {X 0,Y 191.244,Z 308.757,A -85,B 0,C 180,E1 -24687.938,E2 -24687.938} C_VEL
LIN {X 0,Y 195.719,Z 317.892,A -85,B 0,C 180,E1 -24691.107,E2 -24691.107} C_VEL
LIN {X 0,Y 199.951,Z 327.671,A -85,B 0,C 180,E1 -24693.802,E2 -24693.802} C_VEL
LIN {X 0,Y 200.987,Z 330.323,A -85,B 0,C 180,E1 -24694.432,E2 -24694.432} C_VEL
LIN {X 0,Y 195.717,Z 394.761,A -85,B 0,C 180,E1 -24696.272,E2 -24696.272} C_VEL
LIN {X 0,Y 193.528,Z 409.176,A -85,B 0,C 180,E1 -24696.971,E2 -24696.971} C_VEL
LIN {X 0,Y 190.533,Z 422.934,A -85,B 0,C 180,E1 -24697.96,E2 -24697.96} C_VEL
LIN {X 0,Y 186.926,Z 435.498,A -85,B 0,C 180,E1 -24699.153,E2 -24699.153} C_VEL
LIN {X 0,Y 182.104,Z 448.722,A -85,B 0,C 180,E1 -24700.766,E2 -24700.766} C_VEL
LIN {X 0,Y 177.051,Z 461.017,A -85,B 0,C 180,E1 -24702.851,E2 -24702.851} C_VEL
LIN {X 0,Y 171.642,Z 471.777,A -85,B 0,C 180,E1 -24705.064,E2 -24705.064} C_VEL
LIN {X 0,Y 165.41,Z 482.739,A -85,B 0,C 180,E1 -24707.995,E2 -24707.995} C_VEL
LIN {X 0,Y 159.694,Z 491.871,A -85,B 0,C 180,E1 -24711.161,E2 -24711.161} C_VEL
LIN {X 0,Y 154.321,Z 499.518,A -85,B 0,C 180,E1 -24714.503,E2 -24714.503} C_VEL
LIN {X 0,Y 149.783,Z 505.853,A -85,B 0,C 180,E1 -24718.084,E2 -24718.084} C_VEL
LIN {X 0,Y 144.96,Z 512.11,A -85,B 0,C 180,E1 -24722.575,E2 -24722.575} C_VEL
LIN {X 0,Y 140.454,Z 517.667,A -85,B 0,C 180,E1 -24727.957,E2 -24727.957} C_VEL
LIN {X 0,Y 137.929,Z 520.892,A -85,B 0,C 180,E1 -24732.198,E2 -24732.198} C_VEL
LIN {X 0,Y 135.556,Z 523.977,A -85,B 0,C 180,E1 -24738.03,E2 -24738.03} C_VEL
LIN {X 0,Y 134.271,Z 525.804,A -85,B 0,C 180,E1 -24743.99,E2 -24743.99} C_VEL
LIN {X 0,Y 133.867,Z 526.42,A -85,B 0,C 180,E1 -24749.999,E2 -24749.999} C_VEL
LIN {X 0,Y 134.211,Z 525.841,A -85,B 0,C 180,E1 -24756.01,E2 -24756.01} C_VEL
LIN {X 0,Y 135.476,Z 524.057,A -85,B 0,C 180,E1 -24761.975,E2 -24761.975} C_VEL
LIN {X 0,Y 137.864,Z 521.007,A -85,B 0,C 180,E1 -24767.809,E2 -24767.809} C_VEL
LIN {X 0,Y 141.327,Z 516.615,A -85,B 0,C 180,E1 -24773.441,E2 -24773.441} C_VEL
LIN {X 0,Y 146.201,Z 510.734,A -85,B 0,C 180,E1 -24778.73,E2 -24778.73} C_VEL
LIN {X 0,Y 150.91,Z 504.378,A -85,B 0,C 180,E1 -24783.041,E2 -24783.041} C_VEL
LIN {X 0,Y 156.789,Z 496.199,A -85,B 0,C 180,E1 -24787.237,E2 -24787.237} C_VEL
LIN {X 0,Y 163.391,Z 486.363,A -85,B 0,C 180,E1 -24790.99,E2 -24790.99} C_VEL
LIN {X 0,Y 169.419,Z 476.133,A -85,B 0,C 180,E1 -24794.012,E2 -24794.012} C_VEL
LIN {X 0,Y 175.333,Z 464.956,A -85,B 0,C 180,E1 -24796.538,E2 -24796.538} C_VEL
LIN {X 0,Y 180.377,Z 453.679,A -85,B 0,C 180,E1 -24798.589,E2 -24798.589} C_VEL
LIN {X 0,Y 184.976,Z 441.68,A -85,B 0,C 180,E1 -24800.296,E2 -24800.296} C_VEL
LIN {X 0,Y 189.159,Z 428.576,A -85,B 0,C 180,E1 -24801.707,E2 -24801.707} C_VEL
LIN {X 0,Y 192.695,Z 414.509,A -85,B 0,C 180,E1 -24802.813,E2 -24802.813} C_VEL
LIN {X 0,Y 195.28,Z 399.625,A -85,B 0,C 180,E1 -24803.658,E2 -24803.658} C_VEL
LIN {X 0,Y 197.033,Z 383.359,A -85,B 0,C 180,E1 -24804.199,E2 -24804.199} C_VEL
LIN {X 0,Y 201.149,Z 330.459,A -85,B 0,C 180,E1 -24805.709,E2 -24805.709} C_VEL
LIN {X 0,Y 197.262,Z 321.122,A -85,B 0,C 180,E1 -24808.13,E2 -24808.13} C_VEL
LIN {X 0,Y 192.576,Z 311.098,A -85,B 0,C 180,E1 -24811.36,E2 -24811.36} C_VEL
LIN {X 0,Y 188.206,Z 302.889,A -85,B 0,C 180,E1 -24814.803,E2 -24814.803} C_VEL
LIN {X 0,Y 185.431,Z 298.199,A -85,B 0,C 180,E1 -24817.302,E2 -24817.302} C_VEL
LIN {X 0,Y 183.23,Z 294.487,A -85,B 0,C 180,E1 -24819.573,E2 -24819.573} C_VEL
LIN {X 0,Y 180.704,Z 290.381,A -85,B 0,C 180,E1 -24822.618,E2 -24822.618} C_VEL
LIN {X 0,Y 177.619,Z 285.543,A -85,B 0,C 180,E1 -24827.521,E2 -24827.521} C_VEL
LIN {X 0,Y 175.351,Z 282.179,A -85,B 0,C 180,E1 -24833.74,E2 -24833.74} C_VEL
LIN {X 0,Y 174.856,Z 281.091,A -85,B 0,C 180,E1 -24838.848,E2 -24838.848} C_VEL
LIN {X 0,Y 174.998,Z 281.336,A -85,B 0,C 180,E1 -24841.15,E2 -24841.15} C_VEL
LIN {X 0,Y 176.157,Z 283.441,A -85,B 0,C 180,E1 -24846.298,E2 -24846.298} C_VEL
LIN {X 0,Y 178.073,Z 286.175,A -85,B 0,C 180,E1 -24850.517,E2 -24850.517} C_VEL
LIN {X 0,Y 181.473,Z 291.629,A -85,B 0,C 180,E1 -24855.585,E2 -24855.585} C_VEL
LIN {X 0,Y 184.668,Z 296.842,A -85,B 0,C 180,E1 -24859.162,E2 -24859.162} C_VEL
LIN {X 0,Y 187.752,Z 302.177,A -85,B 0,C 180,E1 -24862.056,E2 -24862.056} C_VEL
LIN {X 0,Y 190.949,Z 308.022,A -85,B 0,C 180,E1 -24864.677,E2 -24864.677} C_VEL
LIN {X 0,Y 194.999,Z 316.182,A -85,B 0,C 180,E1 -24867.638,E2 -24867.638} C_VEL
LIN {X 0,Y 199.469,Z 326.362,A -85,B 0,C 180,E1 -24870.576,E2 -24870.576} C_VEL
LIN {X 0,Y 201.287,Z 330.787,A -85,B 0,C 180,E1 -24871.687,E2 -24871.687} C_VEL
LIN {X 0,Y 195.343,Z 400.404,A -85,B 0,C 180,E1 -24873.755,E2 -24873.755} C_VEL
LIN {X 0,Y 192.798,Z 415.693,A -85,B 0,C 180,E1 -24874.44,E2 -24874.44} C_VEL
LIN {X 0,Y 189.256,Z 430.634,A -85,B 0,C 180,E1 -24875.45,E2 -24875.45} C_VEL
LIN {X 0,Y 185.167,Z 444.063,A -85,B 0,C 180,E1 -24876.7,E2 -24876.7} C_VEL
LIN {X 0,Y 180.271,Z 457.217,A -85,B 0,C 180,E1 -24878.32,E2 -24878.32} C_VEL
LIN {X 0,Y 175,Z 469.344,A -85,B 0,C 180,E1 -24880.269,E2 -24880.269} C_VEL
LIN {X 0,Y 169.348,Z 480.592,A -85,B 0,C 180,E1 -24882.557,E2 -24882.557} C_VEL
LIN {X 0,Y 162.98,Z 491.851,A -85,B 0,C 180,E1 -24885.516,E2 -24885.516} C_VEL
LIN {X 0,Y 159.398,Z 497.66,A -85,B 0,C 180,E1 -24887.396,E2 -24887.396} C_VEL
LIN {X 0,Y 156.451,Z 501.52,A -85,B 0,C 180,E1 -24888.656,E2 -24888.656} C_VEL
LIN {X 0,Y 150.264,Z 507.383,A -85,B 0,C 180,E1 -24890.535,E2 -24890.535} C_VEL
LIN {X 0,Y 144.119,Z 512.814,A -85,B 0,C 180,E1 -24892.689,E2 -24892.689} C_VEL
LIN {X 0,Y 141.314,Z 515.849,A -85,B 0,C 180,E1 -24894.371,E2 -24894.371} C_VEL
LIN {X 0,Y 136.361,Z 522.298,A -85,B 0,C 180,E1 -24898.978,E2 -24898.978} C_VEL
LIN {X 0,Y 131.867,Z 528.303,A -85,B 0,C 180,E1 -24904.764,E2 -24904.764} C_VEL
LIN {X 0,Y 128.769,Z 532.857,A -85,B 0,C 180,E1 -24910.886,E2 -24910.886} C_VEL
LIN {X 0,Y 126.929,Z 536.06,A -85,B 0,C 180,E1 -24917.206,E2 -24917.206} C_VEL
LIN {X 0,Y 126.437,Z 537.986,A -85,B 0,C 180,E1 -24923.619,E2 -24923.619} C_VEL
LIN {X 0,Y 126.576,Z 538.548,A -85,B 0,C 180,E1 -24928.051,E2 -24928.051} C_VEL
LIN {X 0,Y 126.683,Z 538.646,A -85,B 0,C 180,E1 -24930.001,E2 -24930.001} C_VEL
LIN {X 0,Y 126.544,Z 538.47,A -85,B 0,C 180,E1 -24933.185,E2 -24933.185} C_VEL
LIN {X 0,Y 126.565,Z 537.149,A -85,B 0,C 180,E1 -24939.59,E2 -24939.59} C_VEL
LIN {X 0,Y 127.663,Z 534.565,A -85,B 0,C 180,E1 -24945.978,E2 -24945.978} C_VEL
LIN {X 0,Y 130.188,Z 530.682,A -85,B 0,C 180,E1 -24952.204,E2 -24952.204} C_VEL
LIN {X 0,Y 133.971,Z 525.391,A -85,B 0,C 180,E1 -24958.174,E2 -24958.174} C_VEL
LIN {X 0,Y 139.096,Z 518.562,A -85,B 0,C 180,E1 -24963.766,E2 -24963.766} C_VEL
LIN {X 0,Y 144.604,Z 511.135,A -85,B 0,C 180,E1 -24968.293,E2 -24968.293} C_VEL
LIN {X 0,Y 150.812,Z 502.139,A -85,B 0,C 180,E1 -24972.51,E2 -24972.51} C_VEL
LIN {X 0,Y 156.881,Z 492.9,A -85,B 0,C 180,E1 -24975.789,E2 -24975.789} C_VEL
LIN {X 0,Y 162.27,Z 483.879,A -85,B 0,C 180,E1 -24978.341,E2 -24978.341} C_VEL
LIN {X 0,Y 168.666,Z 472.163,A -85,B 0,C 180,E1 -24980.902,E2 -24980.902} C_VEL
LIN {X 0,Y 174.221,Z 460.279,A -85,B 0,C 180,E1 -24982.95,E2 -24982.95} C_VEL
LIN {X 0,Y 179.046,Z 448.384,A -85,B 0,C 180,E1 -24984.537,E2 -24984.537} C_VEL
LIN {X 0,Y 183.897,Z 433.959,A -85,B 0,C 180,E1 -24985.979,E2 -24985.979} C_VEL
LIN {X 0,Y 187.702,Z 419.485,A -85,B 0,C 180,E1 -24987.029,E2 -24987.029} C_VEL
LIN {X 0,Y 190.519,Z 404.434,A -85,B 0,C 180,E1 -24987.794,E2 -24987.794} C_VEL
LIN {X 0,Y 192.458,Z 386.231,A -85,B 0,C 180,E1 -24988.416,E2 -24988.416} C_VEL
LIN {X 0,Y 197.009,Z 333.273,A -85,B 0,C 180,E1 -24989.957,E2 -24989.957} C_VEL
LIN {X 0,Y 192.476,Z 322.418,A -85,B 0,C 180,E1 -24993.083,E2 -24993.083} C_VEL
LIN {X 0,Y 188.506,Z 313.908,A -85,B 0,C 180,E1 -24996.154,E2 -24996.154} C_VEL
LIN {X 0,Y 185.37,Z 307.888,A -85,B 0,C 180,E1 -24998.894,E2 -24998.894} C_VEL
LIN {X 0,Y 181.664,Z 301.203,A -85,B 0,C 180,E1 -25002.699,E2 -25002.699} C_VEL
LIN {X 0,Y 179.081,Z 296.89,A -85,B 0,C 180,E1 -25005.947,E2 -25005.947} C_VEL
LIN {X 0,Y 176.33,Z 292.217,A -85,B 0,C 180,E1 -25010.537,E2 -25010.537} C_VEL
LIN {X 0,Y 174.19,Z 288.923,A -85,B 0,C 180,E1 -25016.531,E2 -25016.531} C_VEL
LIN {X 0,Y 173.747,Z 287.774,A -85,B 0,C 180,E1 -25020,E2 -25020} C_VEL
LIN {X 0,Y 174.072,Z 288.744,A -85,B 0,C 180,E1 -25025.793,E2 -25025.793} C_VEL
LIN {X 0,Y 174.983,Z 290.455,A -85,B 0,C 180,E1 -25029.245,E2 -25029.245} C_VEL
LIN {X 0,Y 176.691,Z 292.915,A -85,B 0,C 180,E1 -25033.075,E2 -25033.075} C_VEL
LIN {X 0,Y 179.787,Z 297.986,A -85,B 0,C 180,E1 -25037.875,E2 -25037.875} C_VEL
LIN {X 0,Y 182.716,Z 303.102,A -85,B 0,C 180,E1 -25041.314,E2 -25041.314} C_VEL
LIN {X 0,Y 185.905,Z 308.745,A -85,B 0,C 180,E1 -25044.418,E2 -25044.418} C_VEL
LIN {X 0,Y 189.768,Z 316.476,A -85,B 0,C 180,E1 -25047.674,E2 -25047.674} C_VEL
LIN {X 0,Y 193.47,Z 324.602,A -85,B 0,C 180,E1 -25050.416,E2 -25050.416} C_VEL
LIN {X 0,Y 196.926,Z 333.103,A -85,B 0,C 180,E1 -25052.757,E2 -25052.757} C_VEL
LIN {X 0,Y 192.667,Z 385.848,A -85,B 0,C 180,E1 -25054.264,E2 -25054.264} C_VEL
LIN {X 0,Y 190.873,Z 401.277,A -85,B 0,C 180,E1 -25054.811,E2 -25054.811} C_VEL
LIN {X 0,Y 188.097,Z 415.866,A -85,B 0,C 180,E1 -25055.643,E2 -25055.643} C_VEL
LIN {X 0,Y 184.375,Z 430.084,A -85,B 0,C 180,E1 -25056.824,E2 -25056.824} C_VEL
LIN {X 0,Y 180.042,Z 442.919,A -85,B 0,C 180,E1 -25058.225,E2 -25058.225} C_VEL
LIN {X 0,Y 175.451,Z 454.367,A -85,B 0,C 180,E1 -25059.86,E2 -25059.86} C_VEL
LIN {X 0,Y 170.135,Z 465.776,A -85,B 0,C 180,E1 -25061.965,E2 -25061.965} C_VEL
LIN {X 0,Y 164.443,Z 476.02,A -85,B 0,C 180,E1 -25064.286,E2 -25064.286} C_VEL
LIN {X 0,Y 158.172,Z 486.314,A -85,B 0,C 180,E1 -25067.343,E2 -25067.343} C_VEL
LIN {X 0,Y 152.269,Z 494.893,A -85,B 0,C 180,E1 -25070.607,E2 -25070.607} C_VEL
LIN {X 0,Y 146.016,Z 503.206,A -85,B 0,C 180,E1 -25074.719,E2 -25074.719} C_VEL
LIN {X 0,Y 141.595,Z 509.071,A -85,B 0,C 180,E1 -25078.589,E2 -25078.589} C_VEL
LIN {X 0,Y 136.093,Z 515.421,A -85,B 0,C 180,E1 -25083.962,E2 -25083.962} C_VEL
LIN {X 0,Y 131.992,Z 520.222,A -85,B 0,C 180,E1 -25089.75,E2 -25089.75} C_VEL
LIN {X 0,Y 129.737,Z 522.931,A -85,B 0,C 180,E1 -25094.284,E2 -25094.284} C_VEL
LIN {X 0,Y 127.786,Z 525.377,A -85,B 0,C 180,E1 -25100.502,E2 -25100.502} C_VEL
LIN {X 0,Y 126.89,Z 526.594,A -85,B 0,C 180,E1 -25106.824,E2 -25106.824} C_VEL
LIN {X 0,Y 126.857,Z 526.612,A -85,B 0,C 180,E1 -25113.175,E2 -25113.175} C_VEL
LIN {X 0,Y 127.71,Z 525.435,A -85,B 0,C 180,E1 -25119.501,E2 -25119.501} C_VEL
LIN {X 0,Y 129.685,Z 523.027,A -85,B 0,C 180,E1 -25125.72,E2 -25125.72} C_VEL
LIN {X 0,Y 132.862,Z 519.317,A -85,B 0,C 180,E1 -25131.731,E2 -25131.731} C_VEL
LIN {X 0,Y 137.288,Z 514.205,A -85,B 0,C 180,E1 -25137.432,E2 -25137.432} C_VEL
LIN {X 0,Y 141.448,Z 509.308,A -85,B 0,C 180,E1 -25141.445,E2 -25141.445} C_VEL
LIN {X 0,Y 146.806,Z 502.392,A -85,B 0,C 180,E1 -25145.903,E2 -25145.903} C_VEL
LIN {X 0,Y 152.161,Z 495.234,A -85,B 0,C 180,E1 -25149.424,E2 -25149.424} C_VEL
LIN {X 0,Y 158.113,Z 486.718,A -85,B 0,C 180,E1 -25152.674,E2 -25152.674} C_VEL
LIN {X 0,Y 164.409,Z 476.501,A -85,B 0,C 180,E1 -25155.724,E2 -25155.724} C_VEL
LIN {X 0,Y 170.04,Z 466.34,A -85,B 0,C 180,E1 -25158.068,E2 -25158.068} C_VEL
LIN {X 0,Y 175.772,Z 454.095,A -85,B 0,C 180,E1 -25160.321,E2 -25160.321} C_VEL
LIN {X 0,Y 180.542,Z 442.127,A -85,B 0,C 180,E1 -25162.023,E2 -25162.023} C_VEL
LIN {X 0,Y 184.864,Z 429.082,A -85,B 0,C 180,E1 -25163.426,E2 -25163.426} C_VEL
LIN {X 0,Y 188.659,Z 414.384,A -85,B 0,C 180,E1 -25164.575,E2 -25164.575} C_VEL
LIN {X 0,Y 191.244,Z 400.045,A -85,B 0,C 180,E1 -25165.38,E2 -25165.38} C_VEL
LIN {X 0,Y 193.09,Z 383.381,A -85,B 0,C 180,E1 -25165.935,E2 -25165.935} C_VEL
LIN {X 0,Y 197.124,Z 333.282,A -85,B 0,C 180,E1 -25167.367,E2 -25167.367} C_VEL
LIN {X 0,Y 193.158,Z 323.569,A -85,B 0,C 180,E1 -25170.08,E2 -25170.08} C_VEL
LIN {X 0,Y 189.081,Z 314.804,A -85,B 0,C 180,E1 -25173.175,E2 -25173.175} C_VEL
LIN {X 0,Y 185.726,Z 308.266,A -85,B 0,C 180,E1 -25176.07,E2 -25176.07} C_VEL
LIN {X 0,Y 182.162,Z 301.88,A -85,B 0,C 180,E1 -25179.682,E2 -25179.682} C_VEL
LIN {X 0,Y 179.291,Z 297.027,A -85,B 0,C 180,E1 -25183.271,E2 -25183.271} C_VEL
LIN {X 0,Y 176.413,Z 292.304,A -85,B 0,C 180,E1 -25188.152,E2 -25188.152} C_VEL
LIN {X 0,Y 174.369,Z 289.011,A -85,B 0,C 180,E1 -25194.353,E2 -25194.353} C_VEL
LIN {X 0,Y 174.046,Z 288.098,A -85,B 0,C 180,E1 -25200,E2 -25200} C_VEL
LIN {X 0,Y 175.094,Z 290.28,A -85,B 0,C 180,E1 -25205.759,E2 -25205.759} C_VEL
LIN {X 0,Y 176.892,Z 293.012,A -85,B 0,C 180,E1 -25210.01,E2 -25210.01} C_VEL
LIN {X 0,Y 180.039,Z 298.35,A -85,B 0,C 180,E1 -25214.987,E2 -25214.987} C_VEL
LIN {X 0,Y 182.928,Z 303.277,A -85,B 0,C 180,E1 -25218.406,E2 -25218.406} C_VEL
LIN {X 0,Y 185.808,Z 308.567,A -85,B 0,C 180,E1 -25221.276,E2 -25221.276} C_VEL
LIN {X 0,Y 189.009,Z 314.712,A -85,B 0,C 180,E1 -25224.043,E2 -25224.043} C_VEL
LIN {X 0,Y 193.265,Z 323.916,A -85,B 0,C 180,E1 -25227.302,E2 -25227.302} C_VEL
LIN {X 0,Y 197.205,Z 333.527,A -85,B 0,C 180,E1 -25230.01,E2 -25230.01} C_VEL
LIN {X 0,Y 191.396,Z 400.047,A -85,B 0,C 180,E1 -25232.001,E2 -25232.001} C_VEL
LIN {X 0,Y 188.852,Z 415.052,A -85,B 0,C 180,E1 -25232.653,E2 -25232.653} C_VEL
LIN {X 0,Y 185.218,Z 430.108,A -85,B 0,C 180,E1 -25233.656,E2 -25233.656} C_VEL
LIN {X 0,Y 180.99,Z 443.601,A -85,B 0,C 180,E1 -25234.888,E2 -25234.888} C_VEL
LIN {X 0,Y 175.929,Z 456.797,A -85,B 0,C 180,E1 -25236.493,E2 -25236.493} C_VEL
LIN {X 0,Y 170.484,Z 468.954,A -85,B 0,C 180,E1 -25238.443,E2 -25238.443} C_VEL
LIN {X 0,Y 164.571,Z 480.214,A -85,B 0,C 180,E1 -25240.713,E2 -25240.713} C_VEL
LIN {X 0,Y 157.95,Z 491.492,A -85,B 0,C 180,E1 -25243.696,E2 -25243.696} C_VEL
LIN {X 0,Y 151.795,Z 500.943,A -85,B 0,C 180,E1 -25246.93,E2 -25246.93} C_VEL
LIN {X 0,Y 145.449,Z 510.158,A -85,B 0,C 180,E1 -25251.088,E2 -25251.088} C_VEL
LIN {X 0,Y 141.314,Z 515.849,A -85,B 0,C 180,E1 -25254.371,E2 -25254.371} C_VEL
LIN {X 0,Y 138.547,Z 518.753,A -85,B 0,C 180,E1 -25256.158,E2 -25256.158} C_VEL
LIN {X 0,Y 132.593,Z 523.066,A -85,B 0,C 180,E1 -25258.975,E2 -25258.975} C_VEL
LIN {X 0,Y 126.918,Z 526.851,A -85,B 0,C 180,E1 -25262.158,E2 -25262.158} C_VEL
LIN {X 0,Y 124.684,Z 528.864,A -85,B 0,C 180,E1 -25264.474,E2 -25264.474} C_VEL
LIN {X 0,Y 122,Z 532.52,A -85,B 0,C 180,E1 -25269.781,E2 -25269.781} C_VEL
LIN {X 0,Y 119.96,Z 535.725,A -85,B 0,C 180,E1 -25276.449,E2 -25276.449} C_VEL
LIN {X 0,Y 119.333,Z 537.651,A -85,B 0,C 180,E1 -25283.237,E2 -25283.237} C_VEL
LIN {X 0,Y 119.506,Z 538.255,A -85,B 0,C 180,E1 -25288.697,E2 -25288.697} C_VEL
LIN {X 0,Y 119.517,Z 538.238,A -85,B 0,C 180,E1 -25291.518,E2 -25291.518} C_VEL
LIN {X 0,Y 119.34,Z 537.632,A -85,B 0,C 180,E1 -25296.765,E2 -25296.765} C_VEL
LIN {X 0,Y 119.98,Z 535.68,A -85,B 0,C 180,E1 -25303.552,E2 -25303.552} C_VEL
LIN {X 0,Y 122.028,Z 532.455,A -85,B 0,C 180,E1 -25310.217,E2 -25310.217} C_VEL
LIN {X 0,Y 125.422,Z 527.879,A -85,B 0,C 180,E1 -25316.634,E2 -25316.634} C_VEL
LIN {X 0,Y 130.246,Z 521.836,A -85,B 0,C 180,E1 -25322.657,E2 -25322.657} C_VEL
LIN {X 0,Y 136.483,Z 514.171,A -85,B 0,C 180,E1 -25328.165,E2 -25328.165} C_VEL
LIN {X 0,Y 142.773,Z 505.717,A -85,B 0,C 180,E1 -25332.715,E2 -25332.715} C_VEL
LIN {X 0,Y 149.777,Z 495.829,A -85,B 0,C 180,E1 -25336.662,E2 -25336.662} C_VEL
LIN {X 0,Y 156.432,Z 485.464,A -85,B 0,C 180,E1 -25339.797,E2 -25339.797} C_VEL
LIN {X 0,Y 163.048,Z 474.123,A -85,B 0,C 180,E1 -25342.376,E2 -25342.376} C_VEL
LIN {X 0,Y 169.289,Z 461.511,A -85,B 0,C 180,E1 -25344.624,E2 -25344.624} C_VEL
LIN {X 0,Y 174.347,Z 449.616,A -85,B 0,C 180,E1 -25346.244,E2 -25346.244} C_VEL
LIN {X 0,Y 179.332,Z 435.649,A -85,B 0,C 180,E1 -25347.676,E2 -25347.676} C_VEL
LIN {X 0,Y 183.412,Z 421.107,A -85,B 0,C 180,E1 -25348.757,E2 -25348.757} C_VEL
LIN {X 0,Y 186.496,Z 405.814,A -85,B 0,C 180,E1 -25349.546,E2 -25349.546} C_VEL
LIN {X 0,Y 188.455,Z 389.385,A -85,B 0,C 180,E1 -25350.116,E2 -25350.116} C_VEL
LIN {X 0,Y 193.107,Z 336.163,A -85,B 0,C 180,E1 -25351.689,E2 -25351.689} C_VEL
LIN {X 0,Y 189.041,Z 326.125,A -85,B 0,C 180,E1 -25354.763,E2 -25354.763} C_VEL
LIN {X 0,Y 185.39,Z 318.148,A -85,B 0,C 180,E1 -25357.87,E2 -25357.87} C_VEL
LIN {X 0,Y 182.375,Z 312.117,A -85,B 0,C 180,E1 -25360.807,E2 -25360.807} C_VEL
LIN {X 0,Y 179.719,Z 307.194,A -85,B 0,C 180,E1 -25363.822,E2 -25363.822} C_VEL
LIN {X 0,Y 177.513,Z 303.31,A -85,B 0,C 180,E1 -25366.842,E2 -25366.842} C_VEL
LIN {X 0,Y 175.179,Z 299.036,A -85,B 0,C 180,E1 -25371.057,E2 -25371.057} C_VEL
LIN {X 0,Y 173.26,Z 295.913,A -85,B 0,C 180,E1 -25376.803,E2 -25376.803} C_VEL
LIN {X 0,Y 172.878,Z 294.854,A -85,B 0,C 180,E1 -25380,E2 -25380} C_VEL
LIN {X 0,Y 173.116,Z 295.661,A -85,B 0,C 180,E1 -25385.3,E2 -25385.3} C_VEL
LIN {X 0,Y 173.923,Z 297.296,A -85,B 0,C 180,E1 -25388.716,E2 -25388.716} C_VEL
LIN {X 0,Y 175.456,Z 299.629,A -85,B 0,C 180,E1 -25392.433,E2 -25392.433} C_VEL
LIN {X 0,Y 178.371,Z 304.696,A -85,B 0,C 180,E1 -25397.248,E2 -25397.248} C_VEL
LIN {X 0,Y 180.885,Z 309.297,A -85,B 0,C 180,E1 -25400.394,E2 -25400.394} C_VEL
LIN {X 0,Y 183.775,Z 314.68,A -85,B 0,C 180,E1 -25403.405,E2 -25403.405} C_VEL
LIN {X 0,Y 187.327,Z 322.179,A -85,B 0,C 180,E1 -25406.615,E2 -25406.615} C_VEL
LIN {X 0,Y 190.784,Z 330.153,A -85,B 0,C 180,E1 -25409.36,E2 -25409.36} C_VEL
LIN {X 0,Y 193.11,Z 336.128,A -85,B 0,C 180,E1 -25411.068,E2 -25411.068} C_VEL
LIN {X 0,Y 187.891,Z 395.253,A -85,B 0,C 180,E1 -25412.739,E2 -25412.739} C_VEL
LIN {X 0,Y 185.49,Z 409.952,A -85,B 0,C 180,E1 -25413.447,E2 -25413.447} C_VEL
LIN {X 0,Y 182.186,Z 424.008,A -85,B 0,C 180,E1 -25414.456,E2 -25414.456} C_VEL
LIN {X 0,Y 178.342,Z 436.443,A -85,B 0,C 180,E1 -25415.631,E2 -25415.631} C_VEL
LIN {X 0,Y 173.19,Z 449.57,A -85,B 0,C 180,E1 -25417.216,E2 -25417.216} C_VEL
LIN {X 0,Y 167.578,Z 462.129,A -85,B 0,C 180,E1 -25419.367,E2 -25419.367} C_VEL
LIN {X 0,Y 161.947,Z 472.526,A -85,B 0,C 180,E1 -25421.53,E2 -25421.53} C_VEL
LIN {X 0,Y 155.167,Z 483.459,A -85,B 0,C 180,E1 -25424.49,E2 -25424.49} C_VEL
LIN {X 0,Y 148.904,Z 492.572,A -85,B 0,C 180,E1 -25427.733,E2 -25427.733} C_VEL
LIN {X 0,Y 142.989,Z 500.215,A -85,B 0,C 180,E1 -25431.194,E2 -25431.194} C_VEL
LIN {X 0,Y 137.076,Z 507.594,A -85,B 0,C 180,E1 -25435.668,E2 -25435.668} C_VEL
LIN {X 0,Y 132.511,Z 512.788,A -85,B 0,C 180,E1 -25439.744,E2 -25439.744} C_VEL
LIN {X 0,Y 127.358,Z 518.342,A -85,B 0,C 180,E1 -25445.551,E2 -25445.551} C_VEL
LIN {X 0,Y 124.464,Z 521.56,A -85,B 0,C 180,E1 -25450.195,E2 -25450.195} C_VEL
LIN {X 0,Y 121.677,Z 524.645,A -85,B 0,C 180,E1 -25456.641,E2 -25456.641} C_VEL
LIN {X 0,Y 120.185,Z 526.469,A -85,B 0,C 180,E1 -25463.283,E2 -25463.283} C_VEL
LIN {X 0,Y 119.689,Z 527.085,A -85,B 0,C 180,E1 -25469.999,E2 -25469.999} C_VEL
LIN {X 0,Y 120.112,Z 526.506,A -85,B 0,C 180,E1 -25476.719,E2 -25476.719} C_VEL
LIN {X 0,Y 121.615,Z 524.722,A -85,B 0,C 180,E1 -25483.364,E2 -25483.364} C_VEL
LIN {X 0,Y 124.404,Z 521.673,A -85,B 0,C 180,E1 -25489.812,E2 -25489.812} C_VEL
LIN {X 0,Y 128.401,Z 517.283,A -85,B 0,C 180,E1 -25495.967,E2 -25495.967} C_VEL
LIN {X 0,Y 133.933,Z 511.405,A -85,B 0,C 180,E1 -25501.649,E2 -25501.649} C_VEL
LIN {X 0,Y 138.639,Z 505.725,A -85,B 0,C 180,E1 -25505.797,E2 -25505.797} C_VEL
LIN {X 0,Y 144.773,Z 498.099,A -85,B 0,C 180,E1 -25510.03,E2 -25510.03} C_VEL
LIN {X 0,Y 150.87,Z 490.047,A -85,B 0,C 180,E1 -25513.399,E2 -25513.399} C_VEL
LIN {X 0,Y 157.284,Z 480.453,A -85,B 0,C 180,E1 -25516.559,E2 -25516.559} C_VEL
LIN {X 0,Y 164.166,Z 468.849,A -85,B 0,C 180,E1 -25519.451,E2 -25519.451} C_VEL
LIN {X 0,Y 169.501,Z 458.427,A -85,B 0,C 180,E1 -25521.479,E2 -25521.479} C_VEL
LIN {X 0,Y 175.025,Z 445.718,A -85,B 0,C 180,E1 -25523.423,E2 -25523.423} C_VEL
LIN {X 0,Y 179.478,Z 433.541,A -85,B 0,C 180,E1 -25524.825,E2 -25524.825} C_VEL
LIN {X 0,Y 183.375,Z 420.308,A -85,B 0,C 180,E1 -25525.973,E2 -25525.973} C_VEL
LIN {X 0,Y 186.534,Z 405.653,A -85,B 0,C 180,E1 -25526.91,E2 -25526.91} C_VEL
LIN {X 0,Y 188.499,Z 392.097,A -85,B 0,C 180,E1 -25527.486,E2 -25527.486} C_VEL
LIN {X 0,Y 193.321,Z 336.265,A -85,B 0,C 180,E1 -25529.059,E2 -25529.059} C_VEL
LIN {X 0,Y 189.807,Z 327.532,A -85,B 0,C 180,E1 -25531.679,E2 -25531.679} C_VEL
LIN {X 0,Y 186.076,Z 319.146,A -85,B 0,C 180,E1 -25534.789,E2 -25534.789} C_VEL
LIN {X 0,Y 182.614,Z 312.242,A -85,B 0,C 180,E1 -25538.115,E2 -25538.115} C_VEL
LIN {X 0,Y 179.575,Z 306.725,A -85,B 0,C 180,E1 -25541.606,E2 -25541.606} C_VEL
LIN {X 0,Y 177.797,Z 303.546,A -85,B 0,C 180,E1 -25544.084,E2 -25544.084} C_VEL
LIN {X 0,Y 175.391,Z 299.271,A -85,B 0,C 180,E1 -25548.442,E2 -25548.442} C_VEL
LIN {X 0,Y 173.5,Z 296.125,A -85,B 0,C 180,E1 -25554.325,E2 -25554.325} C_VEL
LIN {X 0,Y 173.178,Z 295.169,A -85,B 0,C 180,E1 -25560,E2 -25560} C_VEL
LIN {X 0,Y 174.046,Z 297.131,A -85,B 0,C 180,E1 -25565.212,E2 -25565.212} C_VEL
LIN {X 0,Y 175.723,Z 299.814,A -85,B 0,C 180,E1 -25569.496,E2 -25569.496} C_VEL
LIN {X 0,Y 178.58,Z 304.954,A -85,B 0,C 180,E1 -25574.311,E2 -25574.311} C_VEL
LIN {X 0,Y 181.1,Z 309.532,A -85,B 0,C 180,E1 -25577.503,E2 -25577.503} C_VEL
LIN {X 0,Y 183.974,Z 315.059,A -85,B 0,C 180,E1 -25580.546,E2 -25580.546} C_VEL
LIN {X 0,Y 187.568,Z 322.485,A -85,B 0,C 180,E1 -25583.805,E2 -25583.805} C_VEL
LIN {X 0,Y 191.384,Z 331.439,A -85,B 0,C 180,E1 -25586.858,E2 -25586.858} C_VEL
LIN {X 0,Y 193.325,Z 336.472,A -85,B 0,C 180,E1 -25588.293,E2 -25588.293} C_VEL
LIN {X 0,Y 187.643,Z 399.697,A -85,B 0,C 180,E1 -25590.179,E2 -25590.179} C_VEL
LIN {X 0,Y 184.939,Z 415.174,A -85,B 0,C 180,E1 -25590.843,E2 -25590.843} C_VEL
LIN {X 0,Y 181.365,Z 429.581,A -85,B 0,C 180,E1 -25591.781,E2 -25591.781} C_VEL
LIN {X 0,Y 177.025,Z 443.143,A -85,B 0,C 180,E1 -25593.002,E2 -25593.002} C_VEL
LIN {X 0,Y 171.775,Z 456.379,A -85,B 0,C 180,E1 -25594.577,E2 -25594.577} C_VEL
LIN {X 0,Y 166.145,Z 468.564,A -85,B 0,C 180,E1 -25596.517,E2 -25596.517} C_VEL
LIN {X 0,Y 160.02,Z 479.839,A -85,B 0,C 180,E1 -25598.781,E2 -25598.781} C_VEL
LIN {X 0,Y 153.081,Z 491.131,A -85,B 0,C 180,E1 -25601.753,E2 -25601.753} C_VEL
LIN {X 0,Y 146.646,Z 500.589,A -85,B 0,C 180,E1 -25605.02,E2 -25605.02} C_VEL
LIN {X 0,Y 139.927,Z 509.811,A -85,B 0,C 180,E1 -25609.238,E2 -25609.238} C_VEL
LIN {X 0,Y 134.849,Z 516.385,A -85,B 0,C 180,E1 -25613.178,E2 -25613.178} C_VEL
LIN {X 0,Y 130.25,Z 521.957,A -85,B 0,C 180,E1 -25617.347,E2 -25617.347} C_VEL
LIN {X 0,Y 125.419,Z 527.966,A -85,B 0,C 180,E1 -25623.368,E2 -25623.368} C_VEL
LIN {X 0,Y 124.684,Z 528.864,A -85,B 0,C 180,E1 -25624.474,E2 -25624.474} C_VEL
LIN {X 0,Y 122.642,Z 530.736,A -85,B 0,C 180,E1 -25626.903,E2 -25626.903} C_VEL
LIN {X 0,Y 117.941,Z 533.288,A -85,B 0,C 180,E1 -25630.885,E2 -25630.885} C_VEL
LIN {X 0,Y 114.419,Z 534.91,A -85,B 0,C 180,E1 -25634.316,E2 -25634.316} C_VEL
LIN {X 0,Y 112.79,Z 535.899,A -85,B 0,C 180,E1 -25637.143,E2 -25637.143} C_VEL
LIN {X 0,Y 112.565,Z 536.178,A -85,B 0,C 180,E1 -25638.127,E2 -25638.127} C_VEL
LIN {X 0,Y 112.242,Z 537.316,A -85,B 0,C 180,E1 -25642.807,E2 -25642.807} C_VEL
LIN {X 0,Y 112.458,Z 537.951,A -85,B 0,C 180,E1 -25649.196,E2 -25649.196} C_VEL
LIN {X 0,Y 112.337,Z 537.802,A -85,B 0,C 180,E1 -25653.588,E2 -25653.588} C_VEL
LIN {X 0,Y 112.467,Z 536.477,A -85,B 0,C 180,E1 -25660.806,E2 -25660.806} C_VEL
LIN {X 0,Y 113.948,Z 533.892,A -85,B 0,C 180,E1 -25667.963,E2 -25667.963} C_VEL
LIN {X 0,Y 116.977,Z 530.003,A -85,B 0,C 180,E1 -25674.871,E2 -25674.871} C_VEL
LIN {X 0,Y 121.482,Z 524.709,A -85,B 0,C 180,E1 -25681.378,E2 -25681.378} C_VEL
LIN {X 0,Y 127.427,Z 517.876,A -85,B 0,C 180,E1 -25687.351,E2 -25687.351} C_VEL
LIN {X 0,Y 133.629,Z 510.439,A -85,B 0,C 180,E1 -25692.111,E2 -25692.111} C_VEL
LIN {X 0,Y 139.51,Z 502.803,A -85,B 0,C 180,E1 -25695.879,E2 -25695.879} C_VEL
LIN {X 0,Y 146.095,Z 493.819,A -85,B 0,C 180,E1 -25699.259,E2 -25699.259} C_VEL
LIN {X 0,Y 153.154,Z 483.123,A -85,B 0,C 180,E1 -25702.333,E2 -25702.333} C_VEL
LIN {X 0,Y 160.037,Z 471.365,A -85,B 0,C 180,E1 -25704.877,E2 -25704.877} C_VEL
LIN {X 0,Y 166.394,Z 458.526,A -85,B 0,C 180,E1 -25707.028,E2 -25707.028} C_VEL
LIN {X 0,Y 171.855,Z 445.669,A -85,B 0,C 180,E1 -25708.615,E2 -25708.615} C_VEL
LIN {X 0,Y 176.651,Z 431.748,A -85,B 0,C 180,E1 -25709.919,E2 -25709.919} C_VEL
LIN {X 0,Y 180.691,Z 416.647,A -85,B 0,C 180,E1 -25710.918,E2 -25710.918} C_VEL
LIN {X 0,Y 183.489,Z 401.514,A -85,B 0,C 180,E1 -25711.612,E2 -25711.612} C_VEL
LIN {X 0,Y 186.005,Z 376.899,A -85,B 0,C 180,E1 -25712.368,E2 -25712.368} C_VEL
LIN {X 0,Y 189.412,Z 339.235,A -85,B 0,C 180,E1 -25713.463,E2 -25713.463} C_VEL
LIN {X 0,Y 186.113,Z 330.776,A -85,B 0,C 180,E1 -25716.198,E2 -25716.198} C_VEL
LIN {X 0,Y 182.797,Z 323.151,A -85,B 0,C 180,E1 -25719.288,E2 -25719.288} C_VEL
LIN {X 0,Y 180.026,Z 317.446,A -85,B 0,C 180,E1 -25722.243,E2 -25722.243} C_VEL
LIN {X 0,Y 177.95,Z 313.375,A -85,B 0,C 180,E1 -25724.832,E2 -25724.832} C_VEL
LIN {X 0,Y 176.077,Z 309.853,A -85,B 0,C 180,E1 -25727.612,E2 -25727.612} C_VEL
LIN {X 0,Y 174.039,Z 305.882,A -85,B 0,C 180,E1 -25731.583,E2 -25731.583} C_VEL
LIN {X 0,Y 172.334,Z 302.903,A -85,B 0,C 180,E1 -25737.078,E2 -25737.078} C_VEL
LIN {X 0,Y 172.008,Z 301.934,A -85,B 0,C 180,E1 -25740,E2 -25740} C_VEL
LIN {X 0,Y 172.251,Z 302.741,A -85,B 0,C 180,E1 -25745.326,E2 -25745.326} C_VEL
LIN {X 0,Y 174.064,Z 305.995,A -85,B 0,C 180,E1 -25751.372,E2 -25751.372} C_VEL
LIN {X 0,Y 176.868,Z 311.167,A -85,B 0,C 180,E1 -25756.447,E2 -25756.447} C_VEL
LIN {X 0,Y 179.401,Z 316.139,A -85,B 0,C 180,E1 -25759.824,E2 -25759.824} C_VEL
LIN {X 0,Y 181.89,Z 321.034,A -85,B 0,C 180,E1 -25762.57,E2 -25762.57} C_VEL
LIN {X 0,Y 185.276,Z 328.571,A -85,B 0,C 180,E1 -25765.817,E2 -25765.817} C_VEL
LIN {X 0,Y 189.047,Z 337.976,A -85,B 0,C 180,E1 -25768.977,E2 -25768.977} C_VEL
LIN {X 0,Y 189.426,Z 338.987,A -85,B 0,C 180,E1 -25769.274,E2 -25769.274} C_VEL
LIN {X 0,Y 184.761,Z 391.406,A -85,B 0,C 180,E1 -25770.744,E2 -25770.744} C_VEL
LIN {X 0,Y 182.624,Z 405.991,A -85,B 0,C 180,E1 -25771.352,E2 -25771.352} C_VEL
LIN {X 0,Y 179.608,Z 419.634,A -85,B 0,C 180,E1 -25772.201,E2 -25772.201} C_VEL
LIN {X 0,Y 175.582,Z 433.062,A -85,B 0,C 180,E1 -25773.325,E2 -25773.325} C_VEL
LIN {X 0,Y 170.953,Z 445.384,A -85,B 0,C 180,E1 -25774.693,E2 -25774.693} C_VEL
LIN {X 0,Y 165.921,Z 456.876,A -85,B 0,C 180,E1 -25776.409,E2 -25776.409} C_VEL
LIN {X 0,Y 159.789,Z 468.707,A -85,B 0,C 180,E1 -25778.675,E2 -25778.675} C_VEL
LIN {X 0,Y 153.717,Z 478.619,A -85,B 0,C 180,E1 -25781.028,E2 -25781.028} C_VEL
LIN {X 0,Y 146.963,Z 488.569,A -85,B 0,C 180,E1 -25784.165,E2 -25784.165} C_VEL
LIN {X 0,Y 140.541,Z 496.919,A -85,B 0,C 180,E1 -25787.538,E2 -25787.538} C_VEL
LIN {X 0,Y 133.776,Z 504.946,A -85,B 0,C 180,E1 -25791.854,E2 -25791.854} C_VEL
LIN {X 0,Y 128.051,Z 511.526,A -85,B 0,C 180,E1 -25796.711,E2 -25796.711} C_VEL
LIN {X 0,Y 122.117,Z 517.467,A -85,B 0,C 180,E1 -25802.585,E2 -25802.585} C_VEL
LIN {X 0,Y 117.807,Z 521.895,A -85,B 0,C 180,E1 -25809.025,E2 -25809.025} C_VEL
LIN {X 0,Y 114.785,Z 524.978,A -85,B 0,C 180,E1 -25815.822,E2 -25815.822} C_VEL
LIN {X 0,Y 113.136,Z 526.803,A -85,B 0,C 180,E1 -25822.862,E2 -25822.862} C_VEL
LIN {X 0,Y 112.607,Z 527.417,A -85,B 0,C 180,E1 -25829.999,E2 -25829.999} C_VEL
LIN {X 0,Y 113.076,Z 526.839,A -85,B 0,C 180,E1 -25837.139,E2 -25837.139} C_VEL
LIN {X 0,Y 114.734,Z 525.054,A -85,B 0,C 180,E1 -25844.181,E2 -25844.181} C_VEL
LIN {X 0,Y 117.752,Z 522.006,A -85,B 0,C 180,E1 -25850.982,E2 -25850.982} C_VEL
LIN {X 0,Y 122.047,Z 517.616,A -85,B 0,C 180,E1 -25857.429,E2 -25857.429} C_VEL
LIN {X 0,Y 127.946,Z 511.741,A -85,B 0,C 180,E1 -25863.317,E2 -25863.317} C_VEL
LIN {X 0,Y 133.085,Z 505.897,A -85,B 0,C 180,E1 -25867.702,E2 -25867.702} C_VEL
LIN {X 0,Y 139.409,Z 498.442,A -85,B 0,C 180,E1 -25871.908,E2 -25871.908} C_VEL
LIN {X 0,Y 145.798,Z 490.398,A -85,B 0,C 180,E1 -25875.314,E2 -25875.314} C_VEL
LIN {X 0,Y 152.486,Z 480.815,A -85,B 0,C 180,E1 -25878.497,E2 -25878.497} C_VEL
LIN {X 0,Y 159.657,Z 469.224,A -85,B 0,C 180,E1 -25881.381,E2 -25881.381} C_VEL
LIN {X 0,Y 165.526,Z 458.109,A -85,B 0,C 180,E1 -25883.528,E2 -25883.528} C_VEL
LIN {X 0,Y 170.904,Z 446.151,A -85,B 0,C 180,E1 -25885.328,E2 -25885.328} C_VEL
LIN {X 0,Y 175.503,Z 434.026,A -85,B 0,C 180,E1 -25886.711,E2 -25886.711} C_VEL
LIN {X 0,Y 179.514,Z 420.88,A -85,B 0,C 180,E1 -25887.843,E2 -25887.843} C_VEL
LIN {X 0,Y 182.72,Z 406.655,A -85,B 0,C 180,E1 -25888.755,E2 -25888.755} C_VEL
LIN {X 0,Y 184.803,Z 393.248,A -85,B 0,C 180,E1 -25889.326,E2 -25889.326} C_VEL
LIN {X 0,Y 189.668,Z 339.314,A -85,B 0,C 180,E1 -25890.827,E2 -25890.827} C_VEL
LIN {X 0,Y 186.234,Z 330.647,A -85,B 0,C 180,E1 -25893.644,E2 -25893.644} C_VEL
LIN {X 0,Y 183.297,Z 323.822,A -85,B 0,C 180,E1 -25896.365,E2 -25896.365} C_VEL
LIN {X 0,Y 180.558,Z 318.085,A -85,B 0,C 180,E1 -25899.248,E2 -25899.248} C_VEL
LIN {X 0,Y 177.849,Z 312.866,A -85,B 0,C 180,E1 -25902.632,E2 -25902.632} C_VEL
LIN {X 0,Y 176.472,Z 310.231,A -85,B 0,C 180,E1 -25904.701,E2 -25904.701} C_VEL
LIN {X 0,Y 174.264,Z 306.126,A -85,B 0,C 180,E1 -25908.955,E2 -25908.955} C_VEL
LIN {X 0,Y 172.543,Z 303.055,A -85,B 0,C 180,E1 -25914.81,E2 -25914.81} C_VEL
LIN {X 0,Y 172.311,Z 302.235,A -85,B 0,C 180,E1 -25920,E2 -25920} C_VEL
LIN {X 0,Y 173.172,Z 304.277,A -85,B 0,C 180,E1 -25925.239,E2 -25925.239} C_VEL
LIN {X 0,Y 174.629,Z 306.781,A -85,B 0,C 180,E1 -25929.122,E2 -25929.122} C_VEL
LIN {X 0,Y 177.14,Z 311.606,A -85,B 0,C 180,E1 -25933.625,E2 -25933.625} C_VEL
LIN {X 0,Y 179.429,Z 315.998,A -85,B 0,C 180,E1 -25936.717,E2 -25936.717} C_VEL
LIN {X 0,Y 182.494,Z 322.157,A -85,B 0,C 180,E1 -25940.132,E2 -25940.132} C_VEL
LIN {X 0,Y 186.003,Z 330.181,A -85,B 0,C 180,E1 -25943.473,E2 -25943.473} C_VEL
LIN {X 0,Y 189.129,Z 338.147,A -85,B 0,C 180,E1 -25946.111,E2 -25946.111} C_VEL
LIN {X 0,Y 189.673,Z 339.644,A -85,B 0,C 180,E1 -25946.548,E2 -25946.548} C_VEL
LIN {X 0,Y 183.965,Z 400.197,A -85,B 0,C 180,E1 -25948.317,E2 -25948.317} C_VEL
LIN {X 0,Y 181.22,Z 415.297,A -85,B 0,C 180,E1 -25948.957,E2 -25948.957} C_VEL
LIN {X 0,Y 177.715,Z 429.055,A -85,B 0,C 180,E1 -25949.828,E2 -25949.828} C_VEL
LIN {X 0,Y 173.25,Z 442.683,A -85,B 0,C 180,E1 -25951.027,E2 -25951.027} C_VEL
LIN {X 0,Y 167.822,Z 455.96,A -85,B 0,C 180,E1 -25952.567,E2 -25952.567} C_VEL
LIN {X 0,Y 161.992,Z 468.172,A -85,B 0,C 180,E1 -25954.484,E2 -25954.484} C_VEL
LIN {X 0,Y 155.657,Z 479.462,A -85,B 0,C 180,E1 -25956.737,E2 -25956.737} C_VEL
LIN {X 0,Y 148.408,Z 490.771,A -85,B 0,C 180,E1 -25959.69,E2 -25959.69} C_VEL
LIN {X 0,Y 141.653,Z 500.233,A -85,B 0,C 180,E1 -25962.964,E2 -25962.964} C_VEL
LIN {X 0,Y 134.55,Z 509.464,A -85,B 0,C 180,E1 -25967.234,E2 -25967.234} C_VEL
LIN {X 0,Y 129.161,Z 516.042,A -85,B 0,C 180,E1 -25971.265,E2 -25971.265} C_VEL
LIN {X 0,Y 122.818,Z 523.269,A -85,B 0,C 180,E1 -25977.072,E2 -25977.072} C_VEL
LIN {X 0,Y 117.894,Z 528.949,A -85,B 0,C 180,E1 -25983.534,E2 -25983.534} C_VEL
LIN {X 0,Y 115.273,Z 532.182,A -85,B 0,C 180,E1 -25988.544,E2 -25988.544} C_VEL
LIN {X 0,Y 113.003,Z 535.389,A -85,B 0,C 180,E1 -25995.597,E2 -25995.597} C_VEL
LIN {X 0,Y 112.565,Z 536.178,A -85,B 0,C 180,E1 -25998.127,E2 -25998.127} C_VEL
LIN {X 0,Y 111.652,Z 536.967,A -85,B 0,C 180,E1 -26001.086,E2 -26001.086} C_VEL
LIN {X 0,Y 110.025,Z 537.487,A -85,B 0,C 180,E1 -26004.032,E2 -26004.032} C_VEL
LIN {X 0,Y 106.409,Z 537.754,A -85,B 0,C 180,E1 -26010.121,E2 -26010.121} C_VEL
LIN {X 0,Y 105.193,Z 537.39,A -85,B 0,C 180,E1 -26014.427,E2 -26014.427} C_VEL
LIN {X 0,Y 105.459,Z 536.141,A -85,B 0,C 180,E1 -26021.534,E2 -26021.534} C_VEL
LIN {X 0,Y 107.157,Z 533.554,A -85,B 0,C 180,E1 -26029.144,E2 -26029.144} C_VEL
LIN {X 0,Y 110.481,Z 529.662,A -85,B 0,C 180,E1 -26036.443,E2 -26036.443} C_VEL
LIN {X 0,Y 115.387,Z 524.367,A -85,B 0,C 180,E1 -26043.243,E2 -26043.243} C_VEL
LIN {X 0,Y 121.804,Z 517.533,A -85,B 0,C 180,E1 -26049.398,E2 -26049.398} C_VEL
LIN {X 0,Y 128.381,Z 510.09,A -85,B 0,C 180,E1 -26054.266,E2 -26054.266} C_VEL
LIN {X 0,Y 135.716,Z 501.074,A -85,B 0,C 180,E1 -26058.667,E2 -26058.667} C_VEL
LIN {X 0,Y 142.724,Z 491.806,A -85,B 0,C 180,E1 -26061.988,E2 -26061.988} C_VEL
LIN {X 0,Y 150.178,Z 480.776,A -85,B 0,C 180,E1 -26064.982,E2 -26064.982} C_VEL
LIN {X 0,Y 157.109,Z 468.975,A -85,B 0,C 180,E1 -26067.411,E2 -26067.411} C_VEL
LIN {X 0,Y 163.367,Z 456.519,A -85,B 0,C 180,E1 -26069.361,E2 -26069.361} C_VEL
LIN {X 0,Y 168.961,Z 443.426,A -85,B 0,C 180,E1 -26070.869,E2 -26070.869} C_VEL
LIN {X 0,Y 173.543,Z 430.077,A -85,B 0,C 180,E1 -26072.049,E2 -26072.049} C_VEL
LIN {X 0,Y 177.53,Z 415.229,A -85,B 0,C 180,E1 -26072.964,E2 -26072.964} C_VEL
LIN {X 0,Y 180.209,Z 400.618,A -85,B 0,C 180,E1 -26073.607,E2 -26073.607} C_VEL
LIN {X 0,Y 184.097,Z 362.158,A -85,B 0,C 180,E1 -26074.708,E2 -26074.708} C_VEL
LIN {X 0,Y 185.901,Z 342.348,A -85,B 0,C 180,E1 -26075.307,E2 -26075.307} C_VEL
LIN {X 0,Y 182.636,Z 333.683,A -85,B 0,C 180,E1 -26078.336,E2 -26078.336} C_VEL
LIN {X 0,Y 179.663,Z 326.767,A -85,B 0,C 180,E1 -26081.469,E2 -26081.469} C_VEL
LIN {X 0,Y 176.729,Z 320.455,A -85,B 0,C 180,E1 -26085.168,E2 -26085.168} C_VEL
LIN {X 0,Y 174.753,Z 316.548,A -85,B 0,C 180,E1 -26088.253,E2 -26088.253} C_VEL
LIN {X 0,Y 172.915,Z 312.717,A -85,B 0,C 180,E1 -26092.116,E2 -26092.116} C_VEL
LIN {X 0,Y 171.364,Z 309.791,A -85,B 0,C 180,E1 -26097.65,E2 -26097.65} C_VEL
LIN {X 0,Y 171.141,Z 308.995,A -85,B 0,C 180,E1 -26100,E2 -26100} C_VEL
LIN {X 0,Y 171.284,Z 309.659,A -85,B 0,C 180,E1 -26104.708,E2 -26104.708} C_VEL
LIN {X 0,Y 171.923,Z 311.157,A -85,B 0,C 180,E1 -26107.931,E2 -26107.931} C_VEL
LIN {X 0,Y 173.176,Z 313.373,A -85,B 0,C 180,E1 -26111.431,E2 -26111.431} C_VEL
LIN {X 0,Y 175.519,Z 317.936,A -85,B 0,C 180,E1 -26115.83,E2 -26115.83} C_VEL
LIN {X 0,Y 177.828,Z 322.724,A -85,B 0,C 180,E1 -26119.105,E2 -26119.105} C_VEL
LIN {X 0,Y 180.305,Z 327.935,A -85,B 0,C 180,E1 -26122,E2 -26122} C_VEL
LIN {X 0,Y 183.41,Z 335.513,A -85,B 0,C 180,E1 -26125.163,E2 -26125.163} C_VEL
LIN {X 0,Y 185.934,Z 342.117,A -85,B 0,C 180,E1 -26127.435,E2 -26127.435} C_VEL
LIN {X 0,Y 180.875,Z 395.583,A -85,B 0,C 180,E1 -26128.917,E2 -26128.917} C_VEL
LIN {X 0,Y 178.317,Z 410.321,A -85,B 0,C 180,E1 -26129.601,E2 -26129.601} C_VEL
LIN {X 0,Y 174.934,Z 423.956,A -85,B 0,C 180,E1 -26130.542,E2 -26130.542} C_VEL
LIN {X 0,Y 170.487,Z 437.379,A -85,B 0,C 180,E1 -26131.764,E2 -26131.764} C_VEL
LIN {X 0,Y 165.015,Z 450.417,A -85,B 0,C 180,E1 -26133.299,E2 -26133.299} C_VEL
LIN {X 0,Y 159.599,Z 461.764,A -85,B 0,C 180,E1 -26135.193,E2 -26135.193} C_VEL
LIN {X 0,Y 152.935,Z 473.272,A -85,B 0,C 180,E1 -26137.56,E2 -26137.56} C_VEL
LIN {X 0,Y 146.755,Z 482.512,A -85,B 0,C 180,E1 -26139.983,E2 -26139.983} C_VEL
LIN {X 0,Y 139.87,Z 491.856,A -85,B 0,C 180,E1 -26143.232,E2 -26143.232} C_VEL
LIN {X 0,Y 132.234,Z 500.91,A -85,B 0,C 180,E1 -26147.34,E2 -26147.34} C_VEL
LIN {X 0,Y 125.518,Z 508.284,A -85,B 0,C 180,E1 -26151.981,E2 -26151.981} C_VEL
LIN {X 0,Y 120.463,Z 513.463,A -85,B 0,C 180,E1 -26156.34,E2 -26156.34} C_VEL
LIN {X 0,Y 114.568,Z 519.013,A -85,B 0,C 180,E1 -26162.607,E2 -26162.607} C_VEL
LIN {X 0,Y 111.209,Z 522.228,A -85,B 0,C 180,E1 -26167.716,E2 -26167.716} C_VEL
LIN {X 0,Y 107.93,Z 525.311,A -85,B 0,C 180,E1 -26174.901,E2 -26174.901} C_VEL
LIN {X 0,Y 106.107,Z 527.135,A -85,B 0,C 180,E1 -26182.386,E2 -26182.386} C_VEL
LIN {X 0,Y 105.53,Z 527.749,A -85,B 0,C 180,E1 -26189.999,E2 -26189.999} C_VEL
LIN {X 0,Y 106.038,Z 527.171,A -85,B 0,C 180,E1 -26197.616,E2 -26197.616} C_VEL
LIN {X 0,Y 107.866,Z 525.386,A -85,B 0,C 180,E1 -26205.105,E2 -26205.105} C_VEL
LIN {X 0,Y 111.16,Z 522.338,A -85,B 0,C 180,E1 -26212.291,E2 -26212.291} C_VEL
LIN {X 0,Y 115.784,Z 517.95,A -85,B 0,C 180,E1 -26219.049,E2 -26219.049} C_VEL
LIN {X 0,Y 122.076,Z 512.076,A -85,B 0,C 180,E1 -26225.147,E2 -26225.147} C_VEL
LIN {X 0,Y 127.358,Z 506.419,A -85,B 0,C 180,E1 -26229.53,E2 -26229.53} C_VEL
LIN {X 0,Y 134.214,Z 498.785,A -85,B 0,C 180,E1 -26233.931,E2 -26233.931} C_VEL
LIN {X 0,Y 140.899,Z 490.748,A -85,B 0,C 180,E1 -26237.366,E2 -26237.366} C_VEL
LIN {X 0,Y 147.886,Z 481.176,A -85,B 0,C 180,E1 -26240.554,E2 -26240.554} C_VEL
LIN {X 0,Y 155.333,Z 469.601,A -85,B 0,C 180,E1 -26243.424,E2 -26243.424} C_VEL
LIN {X 0,Y 161.181,Z 458.979,A -85,B 0,C 180,E1 -26245.469,E2 -26245.469} C_VEL
LIN {X 0,Y 166.978,Z 446.584,A -85,B 0,C 180,E1 -26247.326,E2 -26247.326} C_VEL
LIN {X 0,Y 171.729,Z 434.512,A -85,B 0,C 180,E1 -26248.68,E2 -26248.68} C_VEL
LIN {X 0,Y 175.848,Z 421.453,A -85,B 0,C 180,E1 -26249.797,E2 -26249.797} C_VEL
LIN {X 0,Y 179.231,Z 407.025,A -85,B 0,C 180,E1 -26250.701,E2 -26250.701} C_VEL
LIN {X 0,Y 181.364,Z 393.836,A -85,B 0,C 180,E1 -26251.259,E2 -26251.259} C_VEL
LIN {X 0,Y 186.158,Z 342.343,A -85,B 0,C 180,E1 -26252.688,E2 -26252.688} C_VEL
LIN {X 0,Y 182.754,Z 333.435,A -85,B 0,C 180,E1 -26255.822,E2 -26255.822} C_VEL
LIN {X 0,Y 179.621,Z 326.159,A -85,B 0,C 180,E1 -26259.156,E2 -26259.156} C_VEL
LIN {X 0,Y 176.675,Z 319.998,A -85,B 0,C 180,E1 -26262.939,E2 -26262.939} C_VEL
LIN {X 0,Y 174.99,Z 316.679,A -85,B 0,C 180,E1 -26265.611,E2 -26265.611} C_VEL
LIN {X 0,Y 173.031,Z 312.817,A -85,B 0,C 180,E1 -26269.764,E2 -26269.764} C_VEL
LIN {X 0,Y 171.675,Z 310.149,A -85,B 0,C 180,E1 -26274.784,E2 -26274.784} C_VEL
LIN {X 0,Y 171.394,Z 309.483,A -85,B 0,C 180,E1 -26277.65,E2 -26277.65} C_VEL
LIN {X 0,Y 171.475,Z 309.465,A -85,B 0,C 180,E1 -26280.587,E2 -26280.587} C_VEL
LIN {X 0,Y 172.285,Z 311.451,A -85,B 0,C 180,E1 -26285.266,E2 -26285.266} C_VEL
LIN {X 0,Y 173.429,Z 313.511,A -85,B 0,C 180,E1 -26288.476,E2 -26288.476} C_VEL
LIN {X 0,Y 175.77,Z 318.344,A -85,B 0,C 180,E1 -26292.997,E2 -26292.997} C_VEL
LIN {X 0,Y 177.741,Z 322.331,A -85,B 0,C 180,E1 -26295.847,E2 -26295.847} C_VEL
LIN {X 0,Y 180.636,Z 328.548,A -85,B 0,C 180,E1 -26299.311,E2 -26299.311} C_VEL
LIN {X 0,Y 184.104,Z 337.017,A -85,B 0,C 180,E1 -26302.821,E2 -26302.821} C_VEL
LIN {X 0,Y 186.173,Z 342.727,A -85,B 0,C 180,E1 -26304.706,E2 -26304.706} C_VEL
LIN {X 0,Y 180.633,Z 399.688,A -85,B 0,C 180,E1 -26306.339,E2 -26306.339} C_VEL
LIN {X 0,Y 177.892,Z 414.66,A -85,B 0,C 180,E1 -26306.956,E2 -26306.956} C_VEL
LIN {X 0,Y 173.928,Z 429.661,A -85,B 0,C 180,E1 -26307.885,E2 -26307.885} C_VEL
LIN {X 0,Y 168.987,Z 443.997,A -85,B 0,C 180,E1 -26309.151,E2 -26309.151} C_VEL
LIN {X 0,Y 163.407,Z 456.976,A -85,B 0,C 180,E1 -26310.666,E2 -26310.666} C_VEL
LIN {X 0,Y 156.729,Z 470.149,A -85,B 0,C 180,E1 -26312.78,E2 -26312.78} C_VEL
LIN {X 0,Y 150.193,Z 481.082,A -85,B 0,C 180,E1 -26315.03,E2 -26315.03} C_VEL
LIN {X 0,Y 142.723,Z 492.063,A -85,B 0,C 180,E1 -26318.015,E2 -26318.015} C_VEL
LIN {X 0,Y 135.746,Z 501.287,A -85,B 0,C 180,E1 -26321.351,E2 -26321.351} C_VEL
LIN {X 0,Y 128.374,Z 510.267,A -85,B 0,C 180,E1 -26325.735,E2 -26325.735} C_VEL
LIN {X 0,Y 121.819,Z 517.679,A -85,B 0,C 180,E1 -26330.611,E2 -26330.611} C_VEL
LIN {X 0,Y 115.387,Z 524.475,A -85,B 0,C 180,E1 -26336.76,E2 -26336.76} C_VEL
LIN {X 0,Y 110.475,Z 529.741,A -85,B 0,C 180,E1 -26343.559,E2 -26343.559} C_VEL
LIN {X 0,Y 107.137,Z 533.613,A -85,B 0,C 180,E1 -26350.855,E2 -26350.855} C_VEL
LIN {X 0,Y 105.441,Z 536.175,A -85,B 0,C 180,E1 -26358.467,E2 -26358.467} C_VEL
LIN {X 0,Y 105.235,Z 537.477,A -85,B 0,C 180,E1 -26366.172,E2 -26366.172} C_VEL
LIN {X 0,Y 105.419,Z 537.648,A -85,B 0,C 180,E1 -26370.001,E2 -26370.001} C_VEL
LIN {X 0,Y 105.193,Z 537.39,A -85,B 0,C 180,E1 -26374.427,E2 -26374.427} C_VEL
LIN {X 0,Y 104.465,Z 536.944,A -85,B 0,C 180,E1 -26377.618,E2 -26377.618} C_VEL
LIN {X 0,Y 102.067,Z 535.729,A -85,B 0,C 180,E1 -26382.917,E2 -26382.917} C_VEL
LIN {X 0,Y 100.557,Z 534.406,A -85,B 0,C 180,E1 -26387.285,E2 -26387.285} C_VEL
LIN {X 0,Y 100.539,Z 533.174,A -85,B 0,C 180,E1 -26390.594,E2 -26390.594} C_VEL
LIN {X 0,Y 100.858,Z 532.685,A -85,B 0,C 180,E1 -26391.673,E2 -26391.673} C_VEL
LIN {X 0,Y 104.826,Z 528.616,A -85,B 0,C 180,E1 -26399.358,E2 -26399.358} C_VEL
LIN {X 0,Y 111.025,Z 522.462,A -85,B 0,C 180,E1 -26406.969,E2 -26406.969} C_VEL
LIN {X 0,Y 118.274,Z 515.188,A -85,B 0,C 180,E1 -26413.107,E2 -26413.107} C_VEL
LIN {X 0,Y 125.318,Z 507.446,A -85,B 0,C 180,E1 -26417.874,E2 -26417.874} C_VEL
LIN {X 0,Y 132.288,Z 499.286,A -85,B 0,C 180,E1 -26421.594,E2 -26421.594} C_VEL
LIN {X 0,Y 139.653,Z 489.769,A -85,B 0,C 180,E1 -26424.864,E2 -26424.864} C_VEL
LIN {X 0,Y 147.553,Z 478.365,A -85,B 0,C 180,E1 -26427.72,E2 -26427.72} C_VEL
LIN {X 0,Y 154.977,Z 465.68,A -85,B 0,C 180,E1 -26430.146,E2 -26430.146} C_VEL
LIN {X 0,Y 161.274,Z 453.048,A -85,B 0,C 180,E1 -26431.94,E2 -26431.94} C_VEL
LIN {X 0,Y 167.054,Z 439.134,A -85,B 0,C 180,E1 -26433.379,E2 -26433.379} C_VEL
LIN {X 0,Y 171.458,Z 425.893,A -85,B 0,C 180,E1 -26434.392,E2 -26434.392} C_VEL
LIN {X 0,Y 175.153,Z 411.098,A -85,B 0,C 180,E1 -26435.207,E2 -26435.207} C_VEL
LIN {X 0,Y 177.706,Z 395.589,A -85,B 0,C 180,E1 -26435.779,E2 -26435.779} C_VEL
LIN {X 0,Y 182.596,Z 345.56,A -85,B 0,C 180,E1 -26437.206,E2 -26437.206} C_VEL
LIN {X 0,Y 179.52,Z 337.106,A -85,B 0,C 180,E1 -26440.415,E2 -26440.415} C_VEL
LIN {X 0,Y 176.906,Z 330.81,A -85,B 0,C 180,E1 -26443.558,E2 -26443.558} C_VEL
LIN {X 0,Y 174.763,Z 326.07,A -85,B 0,C 180,E1 -26446.631,E2 -26446.631} C_VEL
LIN {X 0,Y 173.299,Z 322.956,A -85,B 0,C 180,E1 -26449.19,E2 -26449.19} C_VEL
LIN {X 0,Y 171.806,Z 319.524,A -85,B 0,C 180,E1 -26452.656,E2 -26452.656} C_VEL
LIN {X 0,Y 170.453,Z 316.759,A -85,B 0,C 180,E1 -26457.933,E2 -26457.933} C_VEL
LIN {X 0,Y 170.271,Z 316.079,A -85,B 0,C 180,E1 -26460,E2 -26460} C_VEL
LIN {X 0,Y 170.418,Z 316.735,A -85,B 0,C 180,E1 -26464.732,E2 -26464.732} C_VEL
LIN {X 0,Y 171.912,Z 319.79,A -85,B 0,C 180,E1 -26470.499,E2 -26470.499} C_VEL
LIN {X 0,Y 174.194,Z 324.669,A -85,B 0,C 180,E1 -26475.204,E2 -26475.204} C_VEL
LIN {X 0,Y 176.23,Z 329.211,A -85,B 0,C 180,E1 -26478.304,E2 -26478.304} C_VEL
LIN {X 0,Y 178.395,Z 334.088,A -85,B 0,C 180,E1 -26481.029,E2 -26481.029} C_VEL
LIN {X 0,Y 181.465,Z 342.06,A -85,B 0,C 180,E1 -26484.376,E2 -26484.376} C_VEL
LIN {X 0,Y 182.606,Z 345.323,A -85,B 0,C 180,E1 -26485.509,E2 -26485.509} C_VEL
LIN {X 0,Y 178.07,Z 392.57,A -85,B 0,C 180,E1 -26486.79,E2 -26486.79} C_VEL
LIN {X 0,Y 175.686,Z 407.445,A -85,B 0,C 180,E1 -26487.403,E2 -26487.403} C_VEL
LIN {X 0,Y 172.502,Z 420.807,A -85,B 0,C 180,E1 -26488.232,E2 -26488.232} C_VEL
LIN {X 0,Y 168.238,Z 434.056,A -85,B 0,C 180,E1 -26489.304,E2 -26489.304} C_VEL
LIN {X 0,Y 162.651,Z 447.841,A -85,B 0,C 180,E1 -26490.82,E2 -26490.82} C_VEL
LIN {X 0,Y 157.101,Z 459.273,A -85,B 0,C 180,E1 -26492.533,E2 -26492.533} C_VEL
LIN {X 0,Y 150.696,Z 470.532,A -85,B 0,C 180,E1 -26494.716,E2 -26494.716} C_VEL
LIN {X 0,Y 143.569,Z 481.114,A -85,B 0,C 180,E1 -26497.299,E2 -26497.299} C_VEL
LIN {X 0,Y 136.259,Z 490.746,A -85,B 0,C 180,E1 -26500.466,E2 -26500.466} C_VEL
LIN {X 0,Y 128.196,Z 500.044,A -85,B 0,C 180,E1 -26504.545,E2 -26504.545} C_VEL
LIN {X 0,Y 121.248,Z 507.277,A -85,B 0,C 180,E1 -26508.898,E2 -26508.898} C_VEL
LIN {X 0,Y 116.452,Z 512.204,A -85,B 0,C 180,E1 -26512.877,E2 -26512.877} C_VEL
LIN {X 0,Y 109.691,Z 518.138,A -85,B 0,C 180,E1 -26519.164,E2 -26519.164} C_VEL
LIN {X 0,Y 104.665,Z 522.563,A -85,B 0,C 180,E1 -26526.24,E2 -26526.24} C_VEL
LIN {X 0,Y 101.093,Z 525.644,A -85,B 0,C 180,E1 -26533.853,E2 -26533.853} C_VEL
LIN {X 0,Y 99.077,Z 527.468,A -85,B 0,C 180,E1 -26541.843,E2 -26541.843} C_VEL
LIN {X 0,Y 98.438,Z 528.082,A -85,B 0,C 180,E1 -26549.998,E2 -26549.998} C_VEL
LIN {X 0,Y 99.003,Z 527.504,A -85,B 0,C 180,E1 -26558.161,E2 -26558.161} C_VEL
LIN {X 0,Y 101.022,Z 525.719,A -85,B 0,C 180,E1 -26566.156,E2 -26566.156} C_VEL
LIN {X 0,Y 104.62,Z 522.67,A -85,B 0,C 180,E1 -26573.768,E2 -26573.768} C_VEL
LIN {X 0,Y 109.63,Z 518.283,A -85,B 0,C 180,E1 -26580.852,E2 -26580.852} C_VEL
LIN {X 0,Y 116.339,Z 512.411,A -85,B 0,C 180,E1 -26587.162,E2 -26587.162} C_VEL
LIN {X 0,Y 122.386,Z 506.347,A -85,B 0,C 180,E1 -26591.934,E2 -26591.934} C_VEL
LIN {X 0,Y 129.208,Z 499.126,A -85,B 0,C 180,E1 -26596.11,E2 -26596.11} C_VEL
LIN {X 0,Y 136.192,Z 491.098,A -85,B 0,C 180,E1 -26599.563,E2 -26599.563} C_VEL
LIN {X 0,Y 143.492,Z 481.536,A -85,B 0,C 180,E1 -26602.737,E2 -26602.737} C_VEL
LIN {X 0,Y 151.22,Z 469.977,A -85,B 0,C 180,E1 -26605.579,E2 -26605.579} C_VEL
LIN {X 0,Y 157.064,Z 459.793,A -85,B 0,C 180,E1 -26607.523,E2 -26607.523} C_VEL
LIN {X 0,Y 163.271,Z 447.016,A -85,B 0,C 180,E1 -26609.415,E2 -26609.415} C_VEL
LIN {X 0,Y 168.847,Z 433.018,A -85,B 0,C 180,E1 -26610.934,E2 -26610.934} C_VEL
LIN {X 0,Y 173.129,Z 419.421,A -85,B 0,C 180,E1 -26611.993,E2 -26611.993} C_VEL
LIN {X 0,Y 176.285,Z 405.643,A -85,B 0,C 180,E1 -26612.812,E2 -26612.812} C_VEL
LIN {X 0,Y 178.41,Z 391.936,A -85,B 0,C 180,E1 -26613.348,E2 -26613.348} C_VEL
LIN {X 0,Y 182.827,Z 345.531,A -85,B 0,C 180,E1 -26614.615,E2 -26614.615} C_VEL
LIN {X 0,Y 179.689,Z 336.932,A -85,B 0,C 180,E1 -26617.885,E2 -26617.885} C_VEL
LIN {X 0,Y 177.121,Z 330.77,A -85,B 0,C 180,E1 -26620.982,E2 -26620.982} C_VEL
LIN {X 0,Y 174.685,Z 325.432,A -85,B 0,C 180,E1 -26624.542,E2 -26624.542} C_VEL
LIN {X 0,Y 173.484,Z 323.006,A -85,B 0,C 180,E1 -26626.68,E2 -26626.68} C_VEL
LIN {X 0,Y 172.055,Z 319.822,A -85,B 0,C 180,E1 -26630.002,E2 -26630.002} C_VEL
LIN {X 0,Y 170.73,Z 317.082,A -85,B 0,C 180,E1 -26635.277,E2 -26635.277} C_VEL
LIN {X 0,Y 170.53,Z 316.53,A -85,B 0,C 180,E1 -26637.638,E2 -26637.638} C_VEL
LIN {X 0,Y 170.584,Z 316.462,A -85,B 0,C 180,E1 -26640.295,E2 -26640.295} C_VEL
LIN {X 0,Y 171.247,Z 318.277,A -85,B 0,C 180,E1 -26644.708,E2 -26644.708} C_VEL
LIN {X 0,Y 172.337,Z 320.484,A -85,B 0,C 180,E1 -26648.058,E2 -26648.058} C_VEL
LIN {X 0,Y 174.34,Z 324.896,A -85,B 0,C 180,E1 -26652.218,E2 -26652.218} C_VEL
LIN {X 0,Y 176.092,Z 328.696,A -85,B 0,C 180,E1 -26654.961,E2 -26654.961} C_VEL
LIN {X 0,Y 178.643,Z 334.56,A -85,B 0,C 180,E1 -26658.27,E2 -26658.27} C_VEL
LIN {X 0,Y 181.777,Z 342.74,A -85,B 0,C 180,E1 -26661.713,E2 -26661.713} C_VEL
LIN {X 0,Y 182.865,Z 345.913,A -85,B 0,C 180,E1 -26662.806,E2 -26662.806} C_VEL
LIN {X 0,Y 177.391,Z 400.077,A -85,B 0,C 180,E1 -26664.328,E2 -26664.328} C_VEL
LIN {X 0,Y 174.591,Z 414.782,A -85,B 0,C 180,E1 -26664.913,E2 -26664.913} C_VEL
LIN {X 0,Y 170.711,Z 429.135,A -85,B 0,C 180,E1 -26665.77,E2 -26665.77} C_VEL
